// TwinCAT 3 PLC project UnloadRobot
// ProgramVersion: 3.1.4024.0
// libraries:
//   Tc2_EtherCAT, * (Beckhoff Automation GmbH)
//   Tc2_MC2, * (Beckhoff Automation GmbH)
//   Tc2_SerialCom, * (Beckhoff Automation GmbH)
//   Tc2_Standard, * (Beckhoff Automation GmbH)
//   Tc2_System, * (Beckhoff Automation GmbH)
//   Tc2_Utilities, * (Beckhoff Automation GmbH)
//   Tc3_Module, * (Beckhoff Automation GmbH)
// project tree:
//   DUTs/ Angles.TcDUT, Box.TcDUT, DUT.TcDUT, Points.TcDUT, SystemStatus.TcDUT
//   GVLs/ GVL_SerialComunication.TcGVL, Robot_Control_State.TcGVL, Robot_Motor.TcGVL, Robot_Parameter.TcGVL, Robot_Status_Info.TcGVL
//   / PlcTask.TcTTO
//   POUs/ AxisAllCtrl.TcPOU, AxisStatus.TcPOU, AxisStatusReadErrorCode.TcPOU, LedControl.TcPOU, LedLogic.TcPOU, TBoxCtrl.TcPOU, WheelCtrlButtonModeCheck.TcPOU, LeftArmFK.TcPOU, ArmFK_bak.TcPOU, LeftArmWristIK.TcPOU, MoveExtPos.TcPOU, RightArmManualCtrlMove.TcPOU, RightArmFK.TcPOU, LeftArmIK.TcPOU, ArmIK_bak.TcPOU, ArmMove.TcPOU, RightArmIK.TcPOU, LeftArmManualCtrlMove.TcPOU, AxisAbs.TcPOU, AxisCaliHomePos.TcPOU, AxisJog.TcPOU, AxisPowerOn.TcPOU, AxisReset.TcPOU, AxisStop.TcPOU, Gate_Back_Move.TcPOU, GateMove.TcPOU, Gate_Small_Move.TcPOU, MAIN.TcPOU, RightArmWristIK.TcPOU, WheelControl.TcPOU
//   POUs/Serial/ BmsSerial.TcPOU, BmsSerialBackground.TcPOU
// real-time tasks:
//   TASK PlcTask10ms: cycle T#10ms, priority 20, ADS port 350
// motion (NC):
//   TASK NC-Task 1 SAF: cycle T#2ms, priority 4, ADS port 501
//   TASK NC-Task 1 SVB: cycle T#10ms, priority 8, ADS port 511
//   AXIS Axis1_LeftArm_Left (id 3)
//     General: UnitName=°
//     Dynamic: Acceleration=100, Deceleration=150
//     Velo: RefSearch=5, RefSync=5, SlowManual=1, FastManual=5, Maximum=3000
//     OtherSettings: AllowMotionCmdToSlave=true, PulseDistancePos=1, PulseDistanceNeg=1
//     encoder EncType=19
//       EncPara: ScaleFactorNumerator=2.35294117647059, ScaleFactorDenominator=8388608, Offset=122.6484, MaxCount=#xffffffff, ReferenceSystem=1
//     drive DrvType=16
//       DrvPara: MaxCount=#xffffffff, DriveControlDWord=#x00020100
//         Analog: VeloReferenz=3300, TorqueSetpointScale=10, ScaleFactorActTorque=0.1
//         TimeComp: TaskDelayCycles=1
//     controller CtrType=1
//       CtrPara: PriorControlFactor=1
//         PosDiffControl: Enable=false
//         Observer: BandWidth=20
//   AXIS Axis2_LeftArm_Right (id 4)
//     General: UnitName=°
//     Dynamic: Acceleration=100
//     Velo: RefSearch=5, RefSync=5, SlowManual=1, FastManual=5, Maximum=3000
//     OtherSettings: AllowMotionCmdToSlave=true, PulseDistancePos=1, PulseDistanceNeg=1
//     encoder EncType=19
//       EncPara: ScaleFactorNumerator=2.35294117647059, ScaleFactorDenominator=8388608, Offset=68.5837, MaxCount=#xffffffff, ReferenceSystem=1
//     drive DrvType=16
//       DrvPara: MaxCount=#xffffffff, DriveControlDWord=#x00020100
//         Analog: VeloReferenz=3300, TorqueSetpointScale=10, ScaleFactorActTorque=0.1
//         TimeComp: TaskDelayCycles=1
//     controller CtrType=1
//       CtrPara: PriorControlFactor=1
//         PosDiffControl: Enable=false
//         Observer: BandWidth=20
//   AXIS Axis3_LeftArm_Wrist (id 5)
//     General: UnitName=°
//     Dynamic: Acceleration=30
//     Velo: RefSearch=5, RefSync=5, SlowManual=1, FastManual=5, Maximum=3000
//     OtherSettings: AllowMotionCmdToSlave=true, PulseDistancePos=1, PulseDistanceNeg=1
//     encoder EncType=19
//       EncPara: ScaleFactorNumerator=2.97520661157025, ScaleFactorDenominator=8388608, Offset=-19.23, MaxCount=#xffffffff, ReferenceSystem=1
//     drive DrvType=16
//       DrvPara: MaxCount=#xffffffff, DriveControlDWord=#x00020100
//         Analog: VeloReferenz=3300, TorqueSetpointScale=10, ScaleFactorActTorque=0.1
//         TimeComp: TaskDelayCycles=1
//     controller CtrType=1
//       CtrPara: PriorControlFactor=1
//         PosDiffControl: Enable=false
//         Observer: BandWidth=20
//   AXIS Axis4_LeftArm_Lift (id 9)
//     Dynamic: Acceleration=30
//     Velo: RefSearch=5, RefSync=5, SlowManual=1, FastManual=5, Maximum=3000
//     OtherSettings: AllowMotionCmdToSlave=true, PulseDistancePos=1, PulseDistanceNeg=1
//     encoder EncType=19
//       EncPara: ScaleFactorNumerator=6.03, ScaleFactorDenominator=8388608, Offset=-15.1688, MaxCount=#xffffffff, ReferenceSystem=1
//     drive DrvType=16
//       DrvPara: MaxCount=#xffffffff, DriveControlDWord=#x00020100
//         Analog: VeloReferenz=3300, TorqueSetpointScale=10, ScaleFactorActTorque=0.1
//         TimeComp: TaskDelayCycles=1
//     controller CtrType=1
//       CtrPara: PriorControlFactor=1
//         Observer: BandWidth=20
//   AXIS Axis5_RightArm_Left (id 6)
//     General: UnitName=°
//     Dynamic: Acceleration=100, Deceleration=100
//     Velo: RefSearch=5, RefSync=5, SlowManual=1, FastManual=5, Maximum=3000
//     OtherSettings: AllowMotionCmdToSlave=true, PulseDistancePos=1, PulseDistanceNeg=1
//     encoder EncType=19
//       EncPara: ScaleFactorNumerator=2.35294117647059, ScaleFactorDenominator=8388608, Offset=113, MaxCount=#xffffffff, ReferenceSystem=1
//     drive DrvType=16
//       DrvPara: MaxCount=#xffffffff, DriveControlDWord=#x00020100
//         Analog: VeloReferenz=3300, TorqueSetpointScale=10, ScaleFactorActTorque=0.1
//         TimeComp: TaskDelayCycles=1
//     controller CtrType=1
//       CtrPara: PriorControlFactor=1
//         PosDiffControl: Enable=false
//         Observer: BandWidth=20
//   AXIS Axis6_RightArm_Right (id 7)
//     General: UnitName=°
//     Dynamic: Acceleration=100, Deceleration=100
//     Velo: RefSearch=5, RefSync=5, SlowManual=1, FastManual=5, Maximum=3000
//     OtherSettings: AllowMotionCmdToSlave=true, PulseDistancePos=1, PulseDistanceNeg=1
//     encoder EncType=19
//       EncPara: ScaleFactorNumerator=2.35294117647059, ScaleFactorDenominator=8388608, Offset=58, MaxCount=#xffffffff, ReferenceSystem=1
//     drive DrvType=16
//       DrvPara: MaxCount=#xffffffff, DriveControlDWord=#x00020100
//         Analog: VeloReferenz=3300, TorqueSetpointScale=10, ScaleFactorActTorque=0.1
//         TimeComp: TaskDelayCycles=1
//     controller CtrType=1
//       CtrPara: PriorControlFactor=1
//         PosDiffControl: Enable=false
//         Observer: BandWidth=20
//   AXIS Axis7_RightArm_Wrist (id 8)
//     General: UnitName=°
//     Dynamic: Acceleration=30
//     Velo: RefSearch=5, RefSync=5, SlowManual=1, FastManual=5, Maximum=3000
//     OtherSettings: AllowMotionCmdToSlave=true, PulseDistancePos=1, PulseDistanceNeg=1
//     encoder EncType=19
//       EncPara: ScaleFactorNumerator=2.97520661157025, ScaleFactorDenominator=8388608, Offset=24.6504, MaxCount=#xffffffff, ReferenceSystem=1
//     drive DrvType=16
//       DrvPara: MaxCount=#xffffffff, DriveControlDWord=#x00020100
//         Analog: VeloReferenz=3300, TorqueSetpointScale=10, ScaleFactorActTorque=0.1
//         TimeComp: TaskDelayCycles=1
//     controller CtrType=1
//       CtrPara: PriorControlFactor=1
//         Observer: BandWidth=20
//   AXIS Axis8_RightArm_Lift (id 10)
//     Dynamic: Acceleration=30
//     Velo: RefSearch=5, RefSync=5, SlowManual=1, FastManual=5, Maximum=3000
//     OtherSettings: AllowMotionCmdToSlave=true, PulseDistancePos=1, PulseDistanceNeg=1
//     encoder EncType=19
//       EncPara: ScaleFactorNumerator=6.03, ScaleFactorDenominator=8388608, Offset=5.5077, MaxCount=#xffffffff, ReferenceSystem=1
//     drive DrvType=16
//       DrvPara: MaxCount=#xffffffff, DriveControlDWord=#x00020100
//         Analog: VeloReferenz=3300, TorqueSetpointScale=10, ScaleFactorActTorque=0.1
//         TimeComp: TaskDelayCycles=1
//     controller CtrType=1
//       CtrPara: PriorControlFactor=1
//         Observer: BandWidth=20
//   AXIS Axis9_BigGate_Left (id 11)
//     Dynamic: Acceleration=101, Deceleration=109.503, Jerk=510.05
//     Velo: RefSearch=5, RefSync=5, SlowManual=1, FastManual=5
//     OtherSettings: AllowMotionCmdToSlave=true, PulseDistancePos=1, PulseDistanceNeg=1
//     encoder EncType=19
//       EncPara: ScaleFactorNumerator=6.03, ScaleFactorDenominator=8388608, Offset=361.3851, MaxCount=#xffffffff, ReferenceSystem=1
//         SoftEndMinControl: Enable=true, Range=-5
//         SoftEndMaxControl: Enable=true, Range=860
//     drive DrvType=16
//       DrvPara: MaxCount=#xffffffff, DriveControlDWord=#x00020100
//         Analog: TorqueSetpointScale=10, ScaleFactorActTorque=0.1
//         TimeComp: TaskDelayCycles=1
//     controller CtrType=1
//       CtrPara: PriorControlFactor=1
//         Observer: BandWidth=20
//   AXIS Axis10_BigGate_Right (id 12)
//     Dynamic: Acceleration=101, Deceleration=108.497, Jerk=510.05
//     Velo: RefSearch=5, RefSync=5, SlowManual=1, FastManual=5
//     OtherSettings: AllowMotionCmdToSlave=true, PulseDistancePos=1, PulseDistanceNeg=1
//     encoder EncType=19
//       EncPara: ScaleFactorNumerator=6.03, ScaleFactorDenominator=8388608, Offset=-371.0742, MaxCount=#xffffffff, ReferenceSystem=1
//         SoftEndMinControl: Enable=true, Range=-860
//         SoftEndMaxControl: Enable=true, Range=5
//     drive DrvType=16
//       DrvPara: MaxCount=#xffffffff, DriveControlDWord=#x00020100
//         Analog: TorqueSetpointScale=10, ScaleFactorActTorque=0.1
//         TimeComp: TaskDelayCycles=1
//     controller CtrType=1
//       CtrPara: PriorControlFactor=1
//         Observer: BandWidth=20
//   AXIS Axis11_SmallGate_Left (id 13)
//     Dynamic: Acceleration=100
//     Velo: RefSearch=5, RefSync=5, SlowManual=1, FastManual=5
//     OtherSettings: AllowMotionCmdToSlave=true, PulseDistancePos=1, PulseDistanceNeg=1
//     encoder EncType=19
//       EncPara: ScaleFactorNumerator=6.03, ScaleFactorDenominator=8388608, Offset=23.9905, MaxCount=#xffffffff, ReferenceSystem=1
//         SoftEndMinControl: Enable=true, Range=-980
//         SoftEndMaxControl: Enable=true, Range=5
//     drive DrvType=16
//       DrvPara: MaxCount=#xffffffff, DriveControlDWord=#x00020100
//         Analog: TorqueSetpointScale=10, ScaleFactorActTorque=0.1
//         TimeComp: TaskDelayCycles=1
//     controller CtrType=1
//       CtrPara: PriorControlFactor=1
//         Observer: BandWidth=20
//   AXIS Axis12_SmallGate_Right (id 14)
//     Dynamic: Acceleration=100
//     Velo: RefSearch=5, RefSync=5, SlowManual=1, FastManual=5
//     OtherSettings: AllowMotionCmdToSlave=true, PulseDistancePos=1, PulseDistanceNeg=1
//     encoder EncType=19
//       EncPara: ScaleFactorNumerator=6.03, ScaleFactorDenominator=8388608, Offset=-28.5893, MaxCount=#xffffffff, ReferenceSystem=1
//         SoftEndMinControl: Enable=true, Range=-5
//         SoftEndMaxControl: Enable=true, Range=980
//     drive DrvType=16
//       DrvPara: MaxCount=#xffffffff, DriveControlDWord=#x00020100
//         Analog: TorqueSetpointScale=10, ScaleFactorActTorque=0.1
//         TimeComp: TaskDelayCycles=1
//     controller CtrType=1
//       CtrPara: PriorControlFactor=1
//         Observer: BandWidth=20
//   AXIS Axis13_BackGate_Left (id 15)
//     Dynamic: Acceleration=100
//     Velo: RefSearch=5, RefSync=5, SlowManual=1, FastManual=5, Maximum=3000
//     OtherSettings: AllowMotionCmdToSlave=true, PulseDistancePos=1, PulseDistanceNeg=1
//     encoder EncType=19
//       EncPara: ScaleFactorNumerator=5, ScaleFactorDenominator=8388608, Offset=-120.0448, MaxCount=#xffffffff, ReferenceSystem=1
//         SoftEndMinControl: Enable=true, Range=-300
//     drive DrvType=16
//       DrvPara: MaxCount=#xffffffff, DriveControlDWord=#x00020100
//         Analog: VeloReferenz=3300, TorqueSetpointScale=10, ScaleFactorActTorque=0.1
//         TimeComp: TaskDelayCycles=1
//     controller CtrType=1
//       CtrPara: PriorControlFactor=1
//         Observer: BandWidth=20
//   AXIS Axis14_BackGate_Right (id 16)
//     Dynamic: Acceleration=100
//     Velo: RefSearch=5, RefSync=5, SlowManual=1, FastManual=5, Maximum=3000
//     OtherSettings: AllowMotionCmdToSlave=true, PulseDistancePos=1, PulseDistanceNeg=1
//     encoder EncType=19
//       EncPara: ScaleFactorNumerator=5, ScaleFactorDenominator=8388608, Offset=-44.1864, MaxCount=#xffffffff, ReferenceSystem=1
//         SoftEndMinControl: Enable=true, Range=-300
//     drive DrvType=16
//       DrvPara: MaxCount=#xffffffff, DriveControlDWord=#x00020100
//         Analog: VeloReferenz=3300, TorqueSetpointScale=10, ScaleFactorActTorque=0.1
//         TimeComp: TaskDelayCycles=1
//     controller CtrType=1
//       CtrPara: PriorControlFactor=1
//         Observer: BandWidth=20
//   AXIS Axis15_RightWheel_Steer (id 18)
//     General: UnitName=°
//     Velo: RefSearch=2, RefSync=2, SlowManual=5, FastManual=10, Maximum=3000
//     OtherSettings: AllowMotionCmdToSlave=true
//     encoder EncType=19
//       EncPara: ScaleFactorNumerator=1.14285714285714, ScaleFactorDenominator=65535, Offset=-120, MaxCount=#xffffffff, ReferenceSystem=1
//     drive DrvType=16
//       DrvPara: MaxCount=#xffffffff, DriveControlDWord=#x00020000
//         Analog: VeloReferenz=3300, TorqueSetpointScale=10, ScaleFactorActTorque=0.1
//         TimeComp: TaskDelayCycles=1
//     controller CtrType=1
//       CtrPara: PriorControlFactor=1
//         PosDiffControl: Enable=false
//         Observer: BandWidth=20
//   AXIS Axis16_RightWheel_Walk (id 19)
//     Dynamic: AccelerationMaximum=1334, DecelerationMaximum=1334, Acceleration=999.99950000025, Deceleration=999.99950000025, Jerk=1000.00100000175
//     Velo: RefSearch=5, RefSync=5, SlowManual=30, FastManual=60, Maximum=3000
//     OtherSettings: AllowMotionCmdToSlave=true
//     encoder EncType=19
//       EncPara: ScaleFactorNumerator=17.27, ScaleFactorDenominator=65535, MaxCount=#xffffffff
//     drive DrvType=16
//       DrvPara: MaxCount=#xffffffff, DriveControlDWord=#x00020000
//         Analog: VeloReferenz=3300, TorqueSetpointScale=10, ScaleFactorActTorque=0.1
//         TimeComp: TaskDelayCycles=1
//     controller CtrType=1
//       CtrPara: PriorControlFactor=1
//         PosDiffControl: Enable=false
//         Observer: BandWidth=20
//   AXIS Axis17_LeftWheel_Steer (id 20)
//     General: UnitName=°
//     Velo: RefSearch=2, RefSync=2, SlowManual=5, FastManual=10
//     OtherSettings: AllowMotionCmdToSlave=true
//     encoder EncType=19
//       EncPara: ScaleFactorNumerator=1.14285714285714, ScaleFactorDenominator=65535, Offset=-120, MaxCount=#xffffffff, ReferenceSystem=1
//     drive DrvType=16
//       DrvPara: MaxCount=#xffffffff, DriveControlDWord=#x00020000
//         Analog: TorqueSetpointScale=10, ScaleFactorActTorque=0.1
//         TimeComp: TaskDelayCycles=1
//     controller CtrType=1
//       CtrPara: PriorControlFactor=1
//         PosDiffControl: Enable=false
//         Observer: BandWidth=20
//   AXIS Axis18_LeftWheel_Walk (id 21)
//     Dynamic: AccelerationMaximum=1334, DecelerationMaximum=1334, Acceleration=999.998, Deceleration=999.998, Jerk=1000
//     Velo: RefSearch=5, RefSync=5, SlowManual=30, FastManual=60, Maximum=3000
//     OtherSettings: AllowMotionCmdToSlave=true
//     encoder EncType=19
//       EncPara: ScaleFactorNumerator=17.27, ScaleFactorDenominator=65535, MaxCount=#xffffffff
//     drive DrvType=16
//       DrvPara: MaxCount=#xffffffff, DriveControlDWord=#x00020000
//         Analog: VeloReferenz=3300, TorqueSetpointScale=10, ScaleFactorActTorque=0.1
//         TimeComp: TaskDelayCycles=1
//     controller CtrType=1
//       CtrPara: PriorControlFactor=1
//         PosDiffControl: Enable=false
//         Observer: BandWidth=20
//   AXIS Axis01_TestArm_Right (id 1)
//     General: UnitName=°
//     Dynamic: Acceleration=100
//     Velo: Maximum=3000
//     OtherSettings: AllowMotionCmdToSlave=true
//     encoder EncType=1
//       EncPara: ScaleFactorNumerator=360, ScaleFactorDenominator=8388608, Offset=-210.5505, ReferenceSystem=1
//         SoftEndMinControl: Enable=true, Range=-40
//         SoftEndMaxControl: Enable=true, Range=130
//     drive DrvType=5
//       Analog: VeloReferenz=3300, TorqueSetpointScale=10, ScaleFactorActTorque=0.1
//       TimeComp: TaskDelayCycles=1
//     controller CtrType=1
//       CtrPara: PriorControlFactor=1
//         Observer: BandWidth=20
//   AXIS Axis02_TestArm_Left (id 2)
//     General: UnitName=°
//     Dynamic: Acceleration=100.851, Jerk=339.029
//     Velo: Maximum=3000
//     OtherSettings: AllowMotionCmdToSlave=true
//     encoder EncType=19
//       EncPara: ScaleFactorNumerator=360, ScaleFactorDenominator=8388608, Offset=225.616, MaxCount=#xffffffff, ReferenceSystem=1
//         SoftEndMinControl: Enable=true, Range=40
//         SoftEndMaxControl: Enable=true, Range=220
//     drive DrvType=16
//       DrvPara: MaxCount=#xffffffff, DriveControlDWord=#x00000100
//         Analog: VeloReferenz=3300, TorqueSetpointScale=10, ScaleFactorActTorque=0.1
//         TimeComp: TaskDelayCycles=1
//     controller CtrType=1
//       CtrPara: PriorControlFactor=1
//         Observer: BandWidth=20
//   AXIS Axis03_TestArm_Wrist (id 17)
//     General: UnitName=°
//     Dynamic: Acceleration=100.851, Jerk=339.029
//     Velo: Maximum=3000
//     OtherSettings: AllowMotionCmdToSlave=true
//     encoder EncType=19
//       EncPara: ScaleFactorNumerator=360, ScaleFactorDenominator=8388608, Offset=225.616, MaxCount=#xffffffff, ReferenceSystem=1
//         SoftEndMinControl: Enable=true, Range=40
//         SoftEndMaxControl: Enable=true, Range=220
//     drive DrvType=16
//       DrvPara: MaxCount=#xffffffff, DriveControlDWord=#x00000100
//         Analog: VeloReferenz=3300, TorqueSetpointScale=10, ScaleFactorActTorque=0.1
//         TimeComp: TaskDelayCycles=1
//     controller CtrType=1
//       CtrPara: PriorControlFactor=1
//         Observer: BandWidth=20
// I/O:
//   DEVICE Device 3 (EtherCAT), AmsNetId 192.168.1.20.2.1
//     Term 8 (EK1200) [EK1200-5000 EtherCAT Power supply (2A E-Bus)]
//       Term 17 (EL1809) [EL1809 16Ch. Dig. Input 24V, 3ms]
//       Term 18 (EL1809) [EL1809 16Ch. Dig. Input 24V, 3ms]
//       Term 19 (EL1809) [EL1809 16Ch. Dig. Input 24V, 3ms]
//       Term 20 (EL2809) [EL2809 16Ch. Dig. Output 24V, 0.5A]
//       Term 21 (EL2809) [EL2809 16Ch. Dig. Output 24V, 0.5A]
//       Term 24 (EK1110) [EK1110 EtherCAT extension]
//     Drive RightWheel Steer (XMC_ESC) [XMC_ESC]
//     Drive RightWheel Walk (XMC_ESC) [XMC_ESC]
//     Drive LeftWheel Steer (XMC_ESC) [XMC_ESC]
//     Drive LeftWheel Walk (XMC_ESC) [XMC_ESC]
//   DEVICE Device 4 (EtherCAT), AmsNetId 192.168.1.20.5.1
//     Drive BackGate Right(MCDLN35BE) [MCDLN35BE]
//     Drive RightArm Wrist (MBDLN25BE) [MBDLN25BE]
//     Drive RightArm Left (MDDLN55BE) [MDDLN55BE]
//     Drive RightArm Lift (MDDLN55BE) [MDDLN55BE]
//     Drive RightArm Right (MDDLN55BE) [MDDLN55BE]
//     Drive SmallGate Right (MDDLN45BE) [MDDLN45BE]
//     Drive BigGate Right (MDDLN55BE) [MDDLN55BE]
//     Drive BackGate Left (MCDLN35BE) [MCDLN35BE]
//     Drive BigGate Left (MDDLN55BE) [MDDLN55BE]
//     Drive SmallGate Left (MDDLN45BE) [MDDLN45BE]
//     Drive LeftArm Lift (MDDLN55BE) [MDDLN55BE]
//     Drive LeftArm Right (MDDLN55BE) [MDDLN55BE]
//     Drive LeftArm Wrist (MBDLN25BE) [MBDLN25BE]
//     Drive LeftArm Left (MDDLN55BE) [MDDLN55BE]
//   DEVICE Device 5 (COM Port)
//   DEVICE Device 6 (NOV-DP-RAM)
//   DEVICE Device 3 (EtherCAT Automation Protocol), AmsNetId 192.168.1.20.4.1
//   DEVICE Device 7 (USB)
//     Box 1 (CX2100 Power Supply)
// variable links:
//   NC-Task 1 SAF/Axes/Axis10_BigGate_Right <-> Device 4 (EtherCAT)/Drive BigGate Right (MDDLN55BE)
//     Drive/Inputs/In/nDataIn1 <-> Transmit PDO mapping 1/Following error actual value
//     Drive/Inputs/In/nDataIn3[0] <-> Transmit PDO mapping 1/Torque actual value
//     Drive/Inputs/In/nDcOutputTime <-> InfoData/DcOutputShift
//     Drive/Inputs/In/nState1 <-> Transmit PDO mapping 1/Statusword
//     Drive/Inputs/In/nState2 <-> Transmit PDO mapping 1/Statusword @bit 8
//     Drive/Inputs/In/nState4 @bit 1 <-> WcState/InputToggle
//     Drive/Inputs/In/nState4 <-> WcState/WcState
//     Drive/Inputs/In/nState5 <-> Transmit PDO mapping 1/Modes of operation display
//     Drive/Outputs/Out/nCtrl1 <-> Receive PDO mapping 1/Controlword
//     Drive/Outputs/Out/nCtrl2 <-> Receive PDO mapping 1/Controlword @bit 8
//     Drive/Outputs/Out/nCtrl5 <-> Receive PDO mapping 1/Modes of operation
//     Drive/Outputs/Out/nDataOut1 <-> Receive PDO mapping 1/Target position
//     Enc/Inputs/In/nDataIn1 <-> Transmit PDO mapping 1/Position actual value
//     Enc/Inputs/In/nDataIn3 <-> Transmit PDO mapping 1/Touch probe pos1 pos value
//     Enc/Inputs/In/nDcInputTime <-> InfoData/DcInputShift
//     Enc/Inputs/In/nState4 @bit 1 <-> WcState/InputToggle
//     Enc/Inputs/In/nState4 <-> WcState/WcState
//     Enc/Inputs/In/nState5 <-> Transmit PDO mapping 1/Touch probe status
//     Enc/Inputs/In/nState6 <-> Transmit PDO mapping 1/Touch probe status @bit 8
//     Enc/Outputs/Out/nCtrl5 <-> Receive PDO mapping 1/Touch probe function
//     Enc/Outputs/Out/nCtrl6 <-> Receive PDO mapping 1/Touch probe function @bit 8
//   NC-Task 1 SAF/Axes/Axis11_SmallGate_Left <-> Device 4 (EtherCAT)/Drive SmallGate Left (MDDLN45BE)
//     Drive/Inputs/In/nDataIn1 <-> Transmit PDO mapping 1/Following error actual value
//     Drive/Inputs/In/nDataIn3[0] <-> Transmit PDO mapping 1/Torque actual value
//     Drive/Inputs/In/nDcOutputTime <-> InfoData/DcOutputShift
//     Drive/Inputs/In/nState1 <-> Transmit PDO mapping 1/Statusword
//     Drive/Inputs/In/nState2 <-> Transmit PDO mapping 1/Statusword @bit 8
//     Drive/Inputs/In/nState4 @bit 1 <-> WcState/InputToggle
//     Drive/Inputs/In/nState4 <-> WcState/WcState
//     Drive/Inputs/In/nState5 <-> Transmit PDO mapping 1/Modes of operation display
//     Drive/Outputs/Out/nCtrl1 <-> Receive PDO mapping 1/Controlword
//     Drive/Outputs/Out/nCtrl2 <-> Receive PDO mapping 1/Controlword @bit 8
//     Drive/Outputs/Out/nCtrl5 <-> Receive PDO mapping 1/Modes of operation
//     Drive/Outputs/Out/nDataOut1 <-> Receive PDO mapping 1/Target position
//     Enc/Inputs/In/nDataIn1 <-> Transmit PDO mapping 1/Position actual value
//     Enc/Inputs/In/nDataIn3 <-> Transmit PDO mapping 1/Touch probe pos1 pos value
//     Enc/Inputs/In/nDcInputTime <-> InfoData/DcInputShift
//     Enc/Inputs/In/nState4 @bit 1 <-> WcState/InputToggle
//     Enc/Inputs/In/nState4 <-> WcState/WcState
//     Enc/Inputs/In/nState5 <-> Transmit PDO mapping 1/Touch probe status
//     Enc/Inputs/In/nState6 <-> Transmit PDO mapping 1/Touch probe status @bit 8
//     Enc/Outputs/Out/nCtrl5 <-> Receive PDO mapping 1/Touch probe function
//     Enc/Outputs/Out/nCtrl6 <-> Receive PDO mapping 1/Touch probe function @bit 8
//   NC-Task 1 SAF/Axes/Axis12_SmallGate_Right <-> Device 4 (EtherCAT)/Drive SmallGate Right (MDDLN45BE)
//     Drive/Inputs/In/nDataIn1 <-> Transmit PDO mapping 1/Following error actual value
//     Drive/Inputs/In/nDataIn3[0] <-> Transmit PDO mapping 1/Torque actual value
//     Drive/Inputs/In/nDcOutputTime <-> InfoData/DcOutputShift
//     Drive/Inputs/In/nState1 <-> Transmit PDO mapping 1/Statusword
//     Drive/Inputs/In/nState2 <-> Transmit PDO mapping 1/Statusword @bit 8
//     Drive/Inputs/In/nState4 @bit 1 <-> WcState/InputToggle
//     Drive/Inputs/In/nState4 <-> WcState/WcState
//     Drive/Inputs/In/nState5 <-> Transmit PDO mapping 1/Modes of operation display
//     Drive/Outputs/Out/nCtrl1 <-> Receive PDO mapping 1/Controlword
//     Drive/Outputs/Out/nCtrl2 <-> Receive PDO mapping 1/Controlword @bit 8
//     Drive/Outputs/Out/nCtrl5 <-> Receive PDO mapping 1/Modes of operation
//     Drive/Outputs/Out/nDataOut1 <-> Receive PDO mapping 1/Target position
//     Enc/Inputs/In/nDataIn1 <-> Transmit PDO mapping 1/Position actual value
//     Enc/Inputs/In/nDataIn3 <-> Transmit PDO mapping 1/Touch probe pos1 pos value
//     Enc/Inputs/In/nDcInputTime <-> InfoData/DcInputShift
//     Enc/Inputs/In/nState4 @bit 1 <-> WcState/InputToggle
//     Enc/Inputs/In/nState4 <-> WcState/WcState
//     Enc/Inputs/In/nState5 <-> Transmit PDO mapping 1/Touch probe status
//     Enc/Inputs/In/nState6 <-> Transmit PDO mapping 1/Touch probe status @bit 8
//     Enc/Outputs/Out/nCtrl5 <-> Receive PDO mapping 1/Touch probe function
//     Enc/Outputs/Out/nCtrl6 <-> Receive PDO mapping 1/Touch probe function @bit 8
//   NC-Task 1 SAF/Axes/Axis13_BackGate_Left <-> Device 4 (EtherCAT)/Drive BackGate Left (MCDLN35BE)
//     Drive/Inputs/In/nDataIn1 <-> Transmit PDO mapping 1/Following error actual value
//     Drive/Inputs/In/nDataIn3[0] <-> Transmit PDO mapping 1/Torque actual value
//     Drive/Inputs/In/nDcOutputTime <-> InfoData/DcOutputShift
//     Drive/Inputs/In/nState1 <-> Transmit PDO mapping 1/Statusword
//     Drive/Inputs/In/nState2 <-> Transmit PDO mapping 1/Statusword @bit 8
//     Drive/Inputs/In/nState4 @bit 1 <-> WcState/InputToggle
//     Drive/Inputs/In/nState4 <-> WcState/WcState
//     Drive/Inputs/In/nState5 <-> Transmit PDO mapping 1/Modes of operation display
//     Drive/Outputs/Out/nCtrl1 <-> Receive PDO mapping 1/Controlword
//     Drive/Outputs/Out/nCtrl2 <-> Receive PDO mapping 1/Controlword @bit 8
//     Drive/Outputs/Out/nCtrl5 <-> Receive PDO mapping 1/Modes of operation
//     Drive/Outputs/Out/nDataOut1 <-> Receive PDO mapping 1/Target position
//     Enc/Inputs/In/nDataIn1 <-> Transmit PDO mapping 1/Position actual value
//     Enc/Inputs/In/nDataIn3 <-> Transmit PDO mapping 1/Touch probe pos1 pos value
//     Enc/Inputs/In/nDcInputTime <-> InfoData/DcInputShift
//     Enc/Inputs/In/nState4 @bit 1 <-> WcState/InputToggle
//     Enc/Inputs/In/nState4 <-> WcState/WcState
//     Enc/Inputs/In/nState5 <-> Transmit PDO mapping 1/Touch probe status
//     Enc/Inputs/In/nState6 <-> Transmit PDO mapping 1/Touch probe status @bit 8
//     Enc/Outputs/Out/nCtrl5 <-> Receive PDO mapping 1/Touch probe function
//     Enc/Outputs/Out/nCtrl6 <-> Receive PDO mapping 1/Touch probe function @bit 8
//   NC-Task 1 SAF/Axes/Axis14_BackGate_Right <-> Device 4 (EtherCAT)/Drive BackGate Right(MCDLN35BE)
//     Drive/Inputs/In/nDataIn1 <-> Transmit PDO mapping 1/Following error actual value
//     Drive/Inputs/In/nDataIn3[0] <-> Transmit PDO mapping 1/Torque actual value
//     Drive/Inputs/In/nDcOutputTime <-> InfoData/DcOutputShift
//     Drive/Inputs/In/nState1 <-> Transmit PDO mapping 1/Statusword
//     Drive/Inputs/In/nState2 <-> Transmit PDO mapping 1/Statusword @bit 8
//     Drive/Inputs/In/nState4 @bit 1 <-> WcState/InputToggle
//     Drive/Inputs/In/nState4 <-> WcState/WcState
//     Drive/Inputs/In/nState5 <-> Transmit PDO mapping 1/Modes of operation display
//     Drive/Outputs/Out/nCtrl1 <-> Receive PDO mapping 1/Controlword
//     Drive/Outputs/Out/nCtrl2 <-> Receive PDO mapping 1/Controlword @bit 8
//     Drive/Outputs/Out/nCtrl5 <-> Receive PDO mapping 1/Modes of operation
//     Drive/Outputs/Out/nDataOut1 <-> Receive PDO mapping 1/Target position
//     Enc/Inputs/In/nDataIn1 <-> Transmit PDO mapping 1/Position actual value
//     Enc/Inputs/In/nDataIn3 <-> Transmit PDO mapping 1/Touch probe pos1 pos value
//     Enc/Inputs/In/nDcInputTime <-> InfoData/DcInputShift
//     Enc/Inputs/In/nState4 @bit 1 <-> WcState/InputToggle
//     Enc/Inputs/In/nState4 <-> WcState/WcState
//     Enc/Inputs/In/nState5 <-> Transmit PDO mapping 1/Touch probe status
//     Enc/Inputs/In/nState6 <-> Transmit PDO mapping 1/Touch probe status @bit 8
//     Enc/Outputs/Out/nCtrl5 <-> Receive PDO mapping 1/Touch probe function
//     Enc/Outputs/Out/nCtrl6 <-> Receive PDO mapping 1/Touch probe function @bit 8
//   NC-Task 1 SAF/Axes/Axis15_RightWheel_Steer <-> Device 3 (EtherCAT)/Drive RightWheel Steer (XMC_ESC)
//     Drive/Inputs/In/nState1 <-> TxPDO/Statusword
//     Drive/Inputs/In/nState2 <-> TxPDO/Statusword
//     Drive/Outputs/Out/nCtrl1 <-> RxPDO/Controlword
//     Drive/Outputs/Out/nDataOut1 <-> RxPDO/Target_position
//     Enc/Inputs/In/nDataIn1 <-> TxPDO/Position actual angle vaule
//   NC-Task 1 SAF/Axes/Axis16_RightWheel_Walk <-> Device 3 (EtherCAT)/Drive RightWheel Walk (XMC_ESC)
//     Drive/Inputs/In/nState1 <-> TxPDO/Statusword
//     Drive/Inputs/In/nState2 <-> TxPDO/Statusword
//     Drive/Outputs/Out/nCtrl1 <-> RxPDO/Controlword
//     Drive/Outputs/Out/nDataOut1 <-> RxPDO/Target_position
//     Enc/Inputs/In/nDataIn1 <-> TxPDO/Position actual angle vaule
//   NC-Task 1 SAF/Axes/Axis17_LeftWheel_Steer <-> Device 3 (EtherCAT)/Drive LeftWheel Steer (XMC_ESC)
//     Drive/Inputs/In/nState1 <-> TxPDO/Statusword
//     Drive/Inputs/In/nState2 <-> TxPDO/Statusword
//     Drive/Outputs/Out/nCtrl1 <-> RxPDO/Controlword
//     Drive/Outputs/Out/nDataOut1 <-> RxPDO/Target_position
//     Enc/Inputs/In/nDataIn1 <-> TxPDO/Position actual angle vaule
//   NC-Task 1 SAF/Axes/Axis18_LeftWheel_Walk <-> Device 3 (EtherCAT)/Drive LeftWheel Walk (XMC_ESC)
//     Drive/Inputs/In/nState1 <-> TxPDO/Statusword
//     Drive/Inputs/In/nState2 <-> TxPDO/Statusword
//     Drive/Outputs/Out/nCtrl1 <-> RxPDO/Controlword
//     Drive/Outputs/Out/nDataOut1 <-> RxPDO/Target_position
//     Enc/Inputs/In/nDataIn1 <-> TxPDO/Position actual angle vaule
//   NC-Task 1 SAF/Axes/Axis1_LeftArm_Left <-> Device 4 (EtherCAT)/Drive LeftArm Left (MDDLN55BE)
//     Drive/Inputs/In/nDataIn1 <-> Transmit PDO mapping 1/Following error actual value
//     Drive/Inputs/In/nDataIn3[0] <-> Transmit PDO mapping 1/Torque actual value
//     Drive/Inputs/In/nDcOutputTime <-> InfoData/DcOutputShift
//     Drive/Inputs/In/nState1 <-> Transmit PDO mapping 1/Statusword
//     Drive/Inputs/In/nState2 <-> Transmit PDO mapping 1/Statusword @bit 8
//     Drive/Inputs/In/nState4 @bit 1 <-> WcState/InputToggle
//     Drive/Inputs/In/nState4 <-> WcState/WcState
//     Drive/Inputs/In/nState5 <-> Transmit PDO mapping 1/Modes of operation display
//     Drive/Outputs/Out/nCtrl1 <-> Receive PDO mapping 1/Controlword
//     Drive/Outputs/Out/nCtrl2 <-> Receive PDO mapping 1/Controlword @bit 8
//     Drive/Outputs/Out/nCtrl5 <-> Receive PDO mapping 1/Modes of operation
//     Drive/Outputs/Out/nDataOut1 <-> Receive PDO mapping 1/Target position
//     Enc/Inputs/In/nDataIn1 <-> Transmit PDO mapping 1/Position actual value
//     Enc/Inputs/In/nDataIn3 <-> Transmit PDO mapping 1/Touch probe pos1 pos value
//     Enc/Inputs/In/nDcInputTime <-> InfoData/DcInputShift
//     Enc/Inputs/In/nState4 @bit 1 <-> WcState/InputToggle
//     Enc/Inputs/In/nState4 <-> WcState/WcState
//     Enc/Inputs/In/nState5 <-> Transmit PDO mapping 1/Touch probe status
//     Enc/Inputs/In/nState6 <-> Transmit PDO mapping 1/Touch probe status @bit 8
//     Enc/Outputs/Out/nCtrl5 <-> Receive PDO mapping 1/Touch probe function
//     Enc/Outputs/Out/nCtrl6 <-> Receive PDO mapping 1/Touch probe function @bit 8
//   NC-Task 1 SAF/Axes/Axis2_LeftArm_Right <-> Device 4 (EtherCAT)/Drive LeftArm Right (MDDLN55BE)
//     Drive/Inputs/In/nDataIn1 <-> Transmit PDO mapping 1/Following error actual value
//     Drive/Inputs/In/nDataIn3[0] <-> Transmit PDO mapping 1/Torque actual value
//     Drive/Inputs/In/nDcOutputTime <-> InfoData/DcOutputShift
//     Drive/Inputs/In/nState1 <-> Transmit PDO mapping 1/Statusword
//     Drive/Inputs/In/nState2 <-> Transmit PDO mapping 1/Statusword @bit 8
//     Drive/Inputs/In/nState4 @bit 1 <-> WcState/InputToggle
//     Drive/Inputs/In/nState4 <-> WcState/WcState
//     Drive/Inputs/In/nState5 <-> Transmit PDO mapping 1/Modes of operation display
//     Drive/Outputs/Out/nCtrl1 <-> Receive PDO mapping 1/Controlword
//     Drive/Outputs/Out/nCtrl2 <-> Receive PDO mapping 1/Controlword @bit 8
//     Drive/Outputs/Out/nCtrl5 <-> Receive PDO mapping 1/Modes of operation
//     Drive/Outputs/Out/nDataOut1 <-> Receive PDO mapping 1/Target position
//     Enc/Inputs/In/nDataIn1 <-> Transmit PDO mapping 1/Position actual value
//     Enc/Inputs/In/nDataIn3 <-> Transmit PDO mapping 1/Touch probe pos1 pos value
//     Enc/Inputs/In/nDcInputTime <-> InfoData/DcInputShift
//     Enc/Inputs/In/nState4 @bit 1 <-> WcState/InputToggle
//     Enc/Inputs/In/nState4 <-> WcState/WcState
//     Enc/Inputs/In/nState5 <-> Transmit PDO mapping 1/Touch probe status
//     Enc/Inputs/In/nState6 <-> Transmit PDO mapping 1/Touch probe status @bit 8
//     Enc/Outputs/Out/nCtrl5 <-> Receive PDO mapping 1/Touch probe function
//     Enc/Outputs/Out/nCtrl6 <-> Receive PDO mapping 1/Touch probe function @bit 8
//   NC-Task 1 SAF/Axes/Axis3_LeftArm_Wrist <-> Device 4 (EtherCAT)/Drive LeftArm Wrist (MBDLN25BE)
//     Drive/Inputs/In/nDataIn1 <-> Transmit PDO mapping 1/Following error actual value
//     Drive/Inputs/In/nDataIn3[0] <-> Transmit PDO mapping 1/Torque actual value
//     Drive/Inputs/In/nDcOutputTime <-> InfoData/DcOutputShift
//     Drive/Inputs/In/nState1 <-> Transmit PDO mapping 1/Statusword
//     Drive/Inputs/In/nState2 <-> Transmit PDO mapping 1/Statusword @bit 8
//     Drive/Inputs/In/nState4 @bit 1 <-> WcState/InputToggle
//     Drive/Inputs/In/nState4 <-> WcState/WcState
//     Drive/Inputs/In/nState5 <-> Transmit PDO mapping 1/Modes of operation display
//     Drive/Outputs/Out/nCtrl1 <-> Receive PDO mapping 1/Controlword
//     Drive/Outputs/Out/nCtrl2 <-> Receive PDO mapping 1/Controlword @bit 8
//     Drive/Outputs/Out/nCtrl5 <-> Receive PDO mapping 1/Modes of operation
//     Drive/Outputs/Out/nDataOut1 <-> Receive PDO mapping 1/Target position
//     Enc/Inputs/In/nDataIn1 <-> Transmit PDO mapping 1/Position actual value
//     Enc/Inputs/In/nDataIn3 <-> Transmit PDO mapping 1/Touch probe pos1 pos value
//     Enc/Inputs/In/nDcInputTime <-> InfoData/DcInputShift
//     Enc/Inputs/In/nState4 @bit 1 <-> WcState/InputToggle
//     Enc/Inputs/In/nState4 <-> WcState/WcState
//     Enc/Inputs/In/nState5 <-> Transmit PDO mapping 1/Touch probe status
//     Enc/Inputs/In/nState6 <-> Transmit PDO mapping 1/Touch probe status @bit 8
//     Enc/Outputs/Out/nCtrl5 <-> Receive PDO mapping 1/Touch probe function
//     Enc/Outputs/Out/nCtrl6 <-> Receive PDO mapping 1/Touch probe function @bit 8
//   NC-Task 1 SAF/Axes/Axis4_LeftArm_Lift <-> Device 4 (EtherCAT)/Drive LeftArm Lift (MDDLN55BE)
//     Drive/Inputs/In/nDataIn1 <-> Transmit PDO mapping 1/Following error actual value
//     Drive/Inputs/In/nDataIn3[0] <-> Transmit PDO mapping 1/Torque actual value
//     Drive/Inputs/In/nDcOutputTime <-> InfoData/DcOutputShift
//     Drive/Inputs/In/nState1 <-> Transmit PDO mapping 1/Statusword
//     Drive/Inputs/In/nState2 <-> Transmit PDO mapping 1/Statusword @bit 8
//     Drive/Inputs/In/nState4 @bit 1 <-> WcState/InputToggle
//     Drive/Inputs/In/nState4 <-> WcState/WcState
//     Drive/Inputs/In/nState5 <-> Transmit PDO mapping 1/Modes of operation display
//     Drive/Outputs/Out/nCtrl1 <-> Receive PDO mapping 1/Controlword
//     Drive/Outputs/Out/nCtrl2 <-> Receive PDO mapping 1/Controlword @bit 8
//     Drive/Outputs/Out/nCtrl5 <-> Receive PDO mapping 1/Modes of operation
//     Drive/Outputs/Out/nDataOut1 <-> Receive PDO mapping 1/Target position
//     Enc/Inputs/In/nDataIn1 <-> Transmit PDO mapping 1/Position actual value
//     Enc/Inputs/In/nDataIn3 <-> Transmit PDO mapping 1/Touch probe pos1 pos value
//     Enc/Inputs/In/nDcInputTime <-> InfoData/DcInputShift
//     Enc/Inputs/In/nState4 @bit 1 <-> WcState/InputToggle
//     Enc/Inputs/In/nState4 <-> WcState/WcState
//     Enc/Inputs/In/nState5 <-> Transmit PDO mapping 1/Touch probe status
//     Enc/Inputs/In/nState6 <-> Transmit PDO mapping 1/Touch probe status @bit 8
//     Enc/Outputs/Out/nCtrl5 <-> Receive PDO mapping 1/Touch probe function
//     Enc/Outputs/Out/nCtrl6 <-> Receive PDO mapping 1/Touch probe function @bit 8
//   NC-Task 1 SAF/Axes/Axis5_RightArm_Left <-> Device 4 (EtherCAT)/Drive RightArm Left (MDDLN55BE)
//     Drive/Inputs/In/nDataIn1 <-> Transmit PDO mapping 1/Following error actual value
//     Drive/Inputs/In/nDataIn3[0] <-> Transmit PDO mapping 1/Torque actual value
//     Drive/Inputs/In/nDcOutputTime <-> InfoData/DcOutputShift
//     Drive/Inputs/In/nState1 <-> Transmit PDO mapping 1/Statusword
//     Drive/Inputs/In/nState2 <-> Transmit PDO mapping 1/Statusword @bit 8
//     Drive/Inputs/In/nState4 @bit 1 <-> WcState/InputToggle
//     Drive/Inputs/In/nState4 <-> WcState/WcState
//     Drive/Inputs/In/nState5 <-> Transmit PDO mapping 1/Modes of operation display
//     Drive/Outputs/Out/nCtrl1 <-> Receive PDO mapping 1/Controlword
//     Drive/Outputs/Out/nCtrl2 <-> Receive PDO mapping 1/Controlword @bit 8
//     Drive/Outputs/Out/nCtrl5 <-> Receive PDO mapping 1/Modes of operation
//     Drive/Outputs/Out/nDataOut1 <-> Receive PDO mapping 1/Target position
//     Enc/Inputs/In/nDataIn1 <-> Transmit PDO mapping 1/Position actual value
//     Enc/Inputs/In/nDataIn3 <-> Transmit PDO mapping 1/Touch probe pos1 pos value
//     Enc/Inputs/In/nDcInputTime <-> InfoData/DcInputShift
//     Enc/Inputs/In/nState4 @bit 1 <-> WcState/InputToggle
//     Enc/Inputs/In/nState4 <-> WcState/WcState
//     Enc/Inputs/In/nState5 <-> Transmit PDO mapping 1/Touch probe status
//     Enc/Inputs/In/nState6 <-> Transmit PDO mapping 1/Touch probe status @bit 8
//     Enc/Outputs/Out/nCtrl5 <-> Receive PDO mapping 1/Touch probe function
//     Enc/Outputs/Out/nCtrl6 <-> Receive PDO mapping 1/Touch probe function @bit 8
//   NC-Task 1 SAF/Axes/Axis6_RightArm_Right <-> Device 4 (EtherCAT)/Drive RightArm Right (MDDLN55BE)
//     Drive/Inputs/In/nDataIn1 <-> Transmit PDO mapping 1/Following error actual value
//     Drive/Inputs/In/nDataIn3[0] <-> Transmit PDO mapping 1/Torque actual value
//     Drive/Inputs/In/nDcOutputTime <-> InfoData/DcOutputShift
//     Drive/Inputs/In/nState1 <-> Transmit PDO mapping 1/Statusword
//     Drive/Inputs/In/nState2 <-> Transmit PDO mapping 1/Statusword @bit 8
//     Drive/Inputs/In/nState4 @bit 1 <-> WcState/InputToggle
//     Drive/Inputs/In/nState4 <-> WcState/WcState
//     Drive/Inputs/In/nState5 <-> Transmit PDO mapping 1/Modes of operation display
//     Drive/Outputs/Out/nCtrl1 <-> Receive PDO mapping 1/Controlword
//     Drive/Outputs/Out/nCtrl2 <-> Receive PDO mapping 1/Controlword @bit 8
//     Drive/Outputs/Out/nCtrl5 <-> Receive PDO mapping 1/Modes of operation
//     Drive/Outputs/Out/nDataOut1 <-> Receive PDO mapping 1/Target position
//     Enc/Inputs/In/nDataIn1 <-> Transmit PDO mapping 1/Position actual value
//     Enc/Inputs/In/nDataIn3 <-> Transmit PDO mapping 1/Touch probe pos1 pos value
//     Enc/Inputs/In/nDcInputTime <-> InfoData/DcInputShift
//     Enc/Inputs/In/nState4 @bit 1 <-> WcState/InputToggle
//     Enc/Inputs/In/nState4 <-> WcState/WcState
//     Enc/Inputs/In/nState5 <-> Transmit PDO mapping 1/Touch probe status
//     Enc/Inputs/In/nState6 <-> Transmit PDO mapping 1/Touch probe status @bit 8
//     Enc/Outputs/Out/nCtrl5 <-> Receive PDO mapping 1/Touch probe function
//     Enc/Outputs/Out/nCtrl6 <-> Receive PDO mapping 1/Touch probe function @bit 8
//   NC-Task 1 SAF/Axes/Axis7_RightArm_Wrist <-> Device 4 (EtherCAT)/Drive RightArm Wrist (MBDLN25BE)
//     Drive/Inputs/In/nDataIn1 <-> Transmit PDO mapping 1/Following error actual value
//     Drive/Inputs/In/nDataIn3[0] <-> Transmit PDO mapping 1/Torque actual value
//     Drive/Inputs/In/nDcOutputTime <-> InfoData/DcOutputShift
//     Drive/Inputs/In/nState1 <-> Transmit PDO mapping 1/Statusword
//     Drive/Inputs/In/nState2 <-> Transmit PDO mapping 1/Statusword @bit 8
//     Drive/Inputs/In/nState4 @bit 1 <-> WcState/InputToggle
//     Drive/Inputs/In/nState4 <-> WcState/WcState
//     Drive/Inputs/In/nState5 <-> Transmit PDO mapping 1/Modes of operation display
//     Drive/Outputs/Out/nCtrl1 <-> Receive PDO mapping 1/Controlword
//     Drive/Outputs/Out/nCtrl2 <-> Receive PDO mapping 1/Controlword @bit 8
//     Drive/Outputs/Out/nCtrl5 <-> Receive PDO mapping 1/Modes of operation
//     Drive/Outputs/Out/nDataOut1 <-> Receive PDO mapping 1/Target position
//     Enc/Inputs/In/nDataIn1 <-> Transmit PDO mapping 1/Position actual value
//     Enc/Inputs/In/nDataIn3 <-> Transmit PDO mapping 1/Touch probe pos1 pos value
//     Enc/Inputs/In/nDcInputTime <-> InfoData/DcInputShift
//     Enc/Inputs/In/nState4 @bit 1 <-> WcState/InputToggle
//     Enc/Inputs/In/nState4 <-> WcState/WcState
//     Enc/Inputs/In/nState5 <-> Transmit PDO mapping 1/Touch probe status
//     Enc/Inputs/In/nState6 <-> Transmit PDO mapping 1/Touch probe status @bit 8
//     Enc/Outputs/Out/nCtrl5 <-> Receive PDO mapping 1/Touch probe function
//     Enc/Outputs/Out/nCtrl6 <-> Receive PDO mapping 1/Touch probe function @bit 8
//   NC-Task 1 SAF/Axes/Axis8_RightArm_Lift <-> Device 4 (EtherCAT)/Drive RightArm Lift (MDDLN55BE)
//     Drive/Inputs/In/nDataIn1 <-> Transmit PDO mapping 1/Following error actual value
//     Drive/Inputs/In/nDataIn3[0] <-> Transmit PDO mapping 1/Torque actual value
//     Drive/Inputs/In/nDcOutputTime <-> InfoData/DcOutputShift
//     Drive/Inputs/In/nState1 <-> Transmit PDO mapping 1/Statusword
//     Drive/Inputs/In/nState2 <-> Transmit PDO mapping 1/Statusword @bit 8
//     Drive/Inputs/In/nState4 @bit 1 <-> WcState/InputToggle
//     Drive/Inputs/In/nState4 <-> WcState/WcState
//     Drive/Inputs/In/nState5 <-> Transmit PDO mapping 1/Modes of operation display
//     Drive/Outputs/Out/nCtrl1 <-> Receive PDO mapping 1/Controlword
//     Drive/Outputs/Out/nCtrl2 <-> Receive PDO mapping 1/Controlword @bit 8
//     Drive/Outputs/Out/nCtrl5 <-> Receive PDO mapping 1/Modes of operation
//     Drive/Outputs/Out/nDataOut1 <-> Receive PDO mapping 1/Target position
//     Enc/Inputs/In/nDataIn1 <-> Transmit PDO mapping 1/Position actual value
//     Enc/Inputs/In/nDataIn3 <-> Transmit PDO mapping 1/Touch probe pos1 pos value
//     Enc/Inputs/In/nDcInputTime <-> InfoData/DcInputShift
//     Enc/Inputs/In/nState4 @bit 1 <-> WcState/InputToggle
//     Enc/Inputs/In/nState4 <-> WcState/WcState
//     Enc/Inputs/In/nState5 <-> Transmit PDO mapping 1/Touch probe status
//     Enc/Inputs/In/nState6 <-> Transmit PDO mapping 1/Touch probe status @bit 8
//     Enc/Outputs/Out/nCtrl5 <-> Receive PDO mapping 1/Touch probe function
//     Enc/Outputs/Out/nCtrl6 <-> Receive PDO mapping 1/Touch probe function @bit 8
//   NC-Task 1 SAF/Axes/Axis9_BigGate_Left <-> Device 4 (EtherCAT)/Drive BigGate Left (MDDLN55BE)
//     Drive/Inputs/In/nDataIn1 <-> Transmit PDO mapping 1/Following error actual value
//     Drive/Inputs/In/nDataIn3[0] <-> Transmit PDO mapping 1/Torque actual value
//     Drive/Inputs/In/nDcOutputTime <-> InfoData/DcOutputShift
//     Drive/Inputs/In/nState1 <-> Transmit PDO mapping 1/Statusword
//     Drive/Inputs/In/nState2 <-> Transmit PDO mapping 1/Statusword @bit 8
//     Drive/Inputs/In/nState4 @bit 1 <-> WcState/InputToggle
//     Drive/Inputs/In/nState4 <-> WcState/WcState
//     Drive/Inputs/In/nState5 <-> Transmit PDO mapping 1/Modes of operation display
//     Drive/Outputs/Out/nCtrl1 <-> Receive PDO mapping 1/Controlword
//     Drive/Outputs/Out/nCtrl2 <-> Receive PDO mapping 1/Controlword @bit 8
//     Drive/Outputs/Out/nCtrl5 <-> Receive PDO mapping 1/Modes of operation
//     Drive/Outputs/Out/nDataOut1 <-> Receive PDO mapping 1/Target position
//     Enc/Inputs/In/nDataIn1 <-> Transmit PDO mapping 1/Position actual value
//     Enc/Inputs/In/nDataIn3 <-> Transmit PDO mapping 1/Touch probe pos1 pos value
//     Enc/Inputs/In/nDcInputTime <-> InfoData/DcInputShift
//     Enc/Inputs/In/nState4 @bit 1 <-> WcState/InputToggle
//     Enc/Inputs/In/nState4 <-> WcState/WcState
//     Enc/Inputs/In/nState5 <-> Transmit PDO mapping 1/Touch probe status
//     Enc/Inputs/In/nState6 <-> Transmit PDO mapping 1/Touch probe status @bit 8
//     Enc/Outputs/Out/nCtrl5 <-> Receive PDO mapping 1/Touch probe function
//     Enc/Outputs/Out/nCtrl6 <-> Receive PDO mapping 1/Touch probe function @bit 8
//   UnloadRobot/UnloadRobot Instance <-> Device 3 (EtherCAT)/Drive LeftWheel Steer (XMC_ESC)
//     PlcTask Outputs/WheelControl.WheelDriver_ModesOfOperation <-> RxPDO/Modes of operation
//   UnloadRobot/UnloadRobot Instance <-> Device 3 (EtherCAT)/Drive LeftWheel Walk (XMC_ESC)
//     PlcTask Outputs/WheelControl.WheelDriver_ModesOfOperation <-> RxPDO/Modes of operation
//   UnloadRobot/UnloadRobot Instance <-> Device 3 (EtherCAT)/Drive RightWheel Steer (XMC_ESC)
//     PlcTask Outputs/WheelControl.WheelDriver_ModesOfOperation <-> RxPDO/Modes of operation
//   UnloadRobot/UnloadRobot Instance <-> Device 3 (EtherCAT)/Drive RightWheel Walk (XMC_ESC)
//     PlcTask Outputs/WheelControl.WheelDriver_ModesOfOperation <-> RxPDO/Modes of operation
//   UnloadRobot/UnloadRobot Instance <-> Device 3 (EtherCAT)/Term 8 (EK1200)/Term 17 (EL1809)
//     PlcTask Inputs/Robot_Control_State.bEmergencyStopBtn <-> Channel 3/Input
//     PlcTask Inputs/Robot_Control_State.bGreenBtn <-> Channel 4/Input
//     PlcTask Inputs/Robot_Control_State.bRedBtn <-> Channel 6/Input
//     PlcTask Inputs/Robot_Control_State.bRemoteCtrl_1btn <-> Channel 14/Input
//     PlcTask Inputs/Robot_Control_State.bRemoteCtrl_2btn <-> Channel 15/Input
//     PlcTask Inputs/Robot_Control_State.bRemoteCtrl_Down <-> Channel 9/Input
//     PlcTask Inputs/Robot_Control_State.bRemoteCtrl_East <-> Channel 10/Input
//     PlcTask Inputs/Robot_Control_State.bRemoteCtrl_North <-> Channel 13/Input
//     PlcTask Inputs/Robot_Control_State.bRemoteCtrl_Online <-> Channel 7/Input
//     PlcTask Inputs/Robot_Control_State.bRemoteCtrl_South <-> Channel 12/Input
//     PlcTask Inputs/Robot_Control_State.bRemoteCtrl_Up <-> Channel 8/Input
//     PlcTask Inputs/Robot_Control_State.bRemoteCtrl_West <-> Channel 11/Input
//     PlcTask Inputs/Robot_Control_State.bTeachBoxAuto <-> Channel 2/Input
//     PlcTask Inputs/Robot_Control_State.bTeachBoxRemote <-> Channel 1/Input
//     PlcTask Inputs/Robot_Control_State.bYellowBtn <-> Channel 5/Input
//     PlcTask Inputs/Robot_Control_State.b_BackBeltCtrlBoxWarning <-> Channel 16/Input
//   UnloadRobot/UnloadRobot Instance <-> Device 3 (EtherCAT)/Term 8 (EK1200)/Term 18 (EL1809)
//     PlcTask Inputs/Robot_Control_State.bLeftArm_Sucker{1..8}_Completed <-> Channel {1..8}/Input  (8 links)
//     PlcTask Inputs/Robot_Control_State.bRightArm_Sucker{1..8}_Completed <-> Channel {9..16}/Input  (8 links)
//   UnloadRobot/UnloadRobot Instance <-> Device 3 (EtherCAT)/Term 8 (EK1200)/Term 19 (EL1809)
//     PlcTask Inputs/Robot_Control_State.bCrash_Sensor_Back <-> Channel 2/Input
//     PlcTask Inputs/Robot_Control_State.bCrash_Sensor_Front <-> Channel 1/Input
//     PlcTask Inputs/Robot_Control_State.bPumpPhaseSequenceProtectionOK <-> Channel 9/Input
//   UnloadRobot/UnloadRobot Instance <-> Device 3 (EtherCAT)/Term 8 (EK1200)/Term 20 (EL2809)
//     PlcTask Outputs/Robot_Control_State.bAxis_GunTong_Back <-> Channel 10/Output
//     PlcTask Outputs/Robot_Control_State.bAxis_GunTong_Left <-> Channel 11/Output
//     PlcTask Outputs/Robot_Control_State.bAxis_GunTong_Middle <-> Channel 13/Output
//     PlcTask Outputs/Robot_Control_State.bAxis_GunTong_Right <-> Channel 12/Output
//     PlcTask Outputs/Robot_Control_State.bBtnLed_Green_Enable <-> Channel 4/Output
//     PlcTask Outputs/Robot_Control_State.bBtnLed_Red_Enable <-> Channel 6/Output
//     PlcTask Outputs/Robot_Control_State.bBtnLed_Yellow_Enable <-> Channel 5/Output
//     PlcTask Outputs/Robot_Control_State.bFrontLight_Left_Enable <-> Channel 7/Output
//     PlcTask Outputs/Robot_Control_State.bFrontLight_Right_Enable <-> Channel 8/Output
//     PlcTask Outputs/Robot_Control_State.bPumpMotor_Enable <-> Channel 9/Output
//     PlcTask Outputs/Robot_Control_State.bTriColorLed_Green_Enable <-> Channel 1/Output
//     PlcTask Outputs/Robot_Control_State.bTriColorLed_Red_Enable <-> Channel 3/Output
//     PlcTask Outputs/Robot_Control_State.bTriColorLed_Yellow_Enable <-> Channel 2/Output
//   UnloadRobot/UnloadRobot Instance <-> Device 3 (EtherCAT)/Term 8 (EK1200)/Term 21 (EL2809)
//     PlcTask Outputs/Robot_Control_State.bLeftArm_SV{1..8} <-> Channel {1..8}/Output  (8 links)
//     PlcTask Outputs/Robot_Control_State.bRightArm_SV{1..8} <-> Channel {9..16}/Output  (8 links)
//   UnloadRobot/UnloadRobot Instance <-> Device 4 (EtherCAT)/Drive BackGate Left (MCDLN35BE)
//     PlcTask Inputs/Robot_Motor.axis_BackGate_Left_Torque <-> Transmit PDO mapping 1/Torque actual value
//   UnloadRobot/UnloadRobot Instance <-> Device 4 (EtherCAT)/Drive BackGate Right(MCDLN35BE)
//     PlcTask Inputs/Robot_Motor.axis_BackGate_Right_Torque <-> Transmit PDO mapping 1/Torque actual value
//   UnloadRobot/UnloadRobot Instance <-> Device 4 (EtherCAT)/Drive BigGate Left (MDDLN55BE)
//     PlcTask Inputs/Robot_Motor.axis_BigGate_Left_Torque <-> Transmit PDO mapping 1/Torque actual value
//   UnloadRobot/UnloadRobot Instance <-> Device 4 (EtherCAT)/Drive BigGate Right (MDDLN55BE)
//     PlcTask Inputs/Robot_Motor.axis_BigGate_Right_Torque <-> Transmit PDO mapping 1/Torque actual value
//   UnloadRobot/UnloadRobot Instance <-> Device 4 (EtherCAT)/Drive LeftArm Left (MDDLN55BE)
//     PlcTask Inputs/Robot_Motor.axis_LeftArm_Left_Torque <-> Transmit PDO mapping 1/Torque actual value
//   UnloadRobot/UnloadRobot Instance <-> Device 4 (EtherCAT)/Drive LeftArm Lift (MDDLN55BE)
//     PlcTask Inputs/Robot_Motor.axis_LeftArm_Lift_Torque <-> Transmit PDO mapping 1/Torque actual value
//   UnloadRobot/UnloadRobot Instance <-> Device 4 (EtherCAT)/Drive LeftArm Right (MDDLN55BE)
//     PlcTask Inputs/Robot_Motor.axis_LeftArm_Right_Torque <-> Transmit PDO mapping 1/Torque actual value
//   UnloadRobot/UnloadRobot Instance <-> Device 4 (EtherCAT)/Drive LeftArm Wrist (MBDLN25BE)
//     PlcTask Inputs/Robot_Motor.axis_LeftArm_Wrist_Torque <-> Transmit PDO mapping 1/Torque actual value
//   UnloadRobot/UnloadRobot Instance <-> Device 4 (EtherCAT)/Drive RightArm Left (MDDLN55BE)
//     PlcTask Inputs/Robot_Motor.axis_RightArm_Left_Torque <-> Transmit PDO mapping 1/Torque actual value
//   UnloadRobot/UnloadRobot Instance <-> Device 4 (EtherCAT)/Drive RightArm Lift (MDDLN55BE)
//     PlcTask Inputs/Robot_Motor.axis_RightArm_Lift_Torque <-> Transmit PDO mapping 1/Torque actual value
//   UnloadRobot/UnloadRobot Instance <-> Device 4 (EtherCAT)/Drive RightArm Right (MDDLN55BE)
//     PlcTask Inputs/Robot_Motor.axis_RightArm_Right_Torque <-> Transmit PDO mapping 1/Torque actual value
//   UnloadRobot/UnloadRobot Instance <-> Device 4 (EtherCAT)/Drive RightArm Wrist (MBDLN25BE)
//     PlcTask Inputs/Robot_Motor.axis_RightArm_Wrist_Torque <-> Transmit PDO mapping 1/Torque actual value
//   UnloadRobot/UnloadRobot Instance <-> Device 4 (EtherCAT)/Drive SmallGate Left (MDDLN45BE)
//     PlcTask Inputs/Robot_Motor.axis_SmallGate_Left_Torque <-> Transmit PDO mapping 1/Torque actual value
//   UnloadRobot/UnloadRobot Instance <-> Device 4 (EtherCAT)/Drive SmallGate Right (MDDLN45BE)
//     PlcTask Inputs/Robot_Motor.axis_SmallGate_Right_Torque <-> Transmit PDO mapping 1/Torque actual value
//   UnloadRobot/UnloadRobot Instance <-> Device 5 (COM Port)
//     PlcTask Inputs/GVL_SerialComunication.pComIn/D[{0..63}] <-> Inputs/Data{1..64}  (64 links)
//     PlcTask Inputs/GVL_SerialComunication.pComIn/SerStatus <-> Inputs/Status
//     PlcTask Outputs/GVL_SerialComunication.pComOut/D[{0..63}] <-> Outputs/Data{1..64}  (64 links)
//     PlcTask Outputs/GVL_SerialComunication.pComOut/SerCtrl <-> Outputs/Ctrl
//   UnloadRobot/UnloadRobot Instance <-> NC-Task 1 SAF/Axes/Axis10_BigGate_Right
//     PlcTask Inputs/Robot_Motor.axis_BigGate_Right.NcToPlc <-> Outputs/ToPlc
//     PlcTask Inputs/Robot_Status_Info.bDriverDeviceErrorCode_axis_BigGate_Right <-> Outputs/ToPlc/ErrorCode
//     PlcTask Inputs/Robot_Status_Info.bDriverDeviceError_axis_BigGate_Right <-> Outputs/ToPlc/StateDWord/DriveDeviceError
//     PlcTask Outputs/Robot_Motor.axis_BigGate_Right.PlcToNc <-> Inputs/FromPlc
//   UnloadRobot/UnloadRobot Instance <-> NC-Task 1 SAF/Axes/Axis11_SmallGate_Left
//     PlcTask Inputs/Robot_Motor.axis_SmallGate_Left.NcToPlc <-> Outputs/ToPlc
//     PlcTask Inputs/Robot_Status_Info.bDriverDeviceErrorCode_axis_SmallGate_Left <-> Outputs/ToPlc/ErrorCode
//     PlcTask Inputs/Robot_Status_Info.bDriverDeviceError_axis_SmallGate_Left <-> Outputs/ToPlc/StateDWord/DriveDeviceError
//     PlcTask Outputs/Robot_Motor.axis_SmallGate_Left.PlcToNc <-> Inputs/FromPlc
//   UnloadRobot/UnloadRobot Instance <-> NC-Task 1 SAF/Axes/Axis12_SmallGate_Right
//     PlcTask Inputs/Robot_Motor.axis_SmallGate_Right.NcToPlc <-> Outputs/ToPlc
//     PlcTask Inputs/Robot_Status_Info.bDriverDeviceErrorCode_axis_SmallGate_Right <-> Outputs/ToPlc/ErrorCode
//     PlcTask Inputs/Robot_Status_Info.bDriverDeviceError_axis_SmallGate_Right <-> Outputs/ToPlc/StateDWord/DriveDeviceError
//     PlcTask Outputs/Robot_Motor.axis_SmallGate_Right.PlcToNc <-> Inputs/FromPlc
//   UnloadRobot/UnloadRobot Instance <-> NC-Task 1 SAF/Axes/Axis13_BackGate_Left
//     PlcTask Inputs/Robot_Motor.axis_BackGate_Left.NcToPlc <-> Outputs/ToPlc
//     PlcTask Inputs/Robot_Status_Info.bDriverDeviceErrorCode_axis_BackGate_Left <-> Outputs/ToPlc/ErrorCode
//     PlcTask Inputs/Robot_Status_Info.bDriverDeviceError_axis_BackGate_Left <-> Outputs/ToPlc/StateDWord/DriveDeviceError
//     PlcTask Outputs/Robot_Motor.axis_BackGate_Left.PlcToNc <-> Inputs/FromPlc
//   UnloadRobot/UnloadRobot Instance <-> NC-Task 1 SAF/Axes/Axis14_BackGate_Right
//     PlcTask Inputs/Robot_Motor.axis_BackGate_Right.NcToPlc <-> Outputs/ToPlc
//     PlcTask Inputs/Robot_Status_Info.bDriverDeviceErrorCode_axis_BackGate_Right <-> Outputs/ToPlc/ErrorCode
//     PlcTask Inputs/Robot_Status_Info.bDriverDeviceError_axis_BackGate_Right <-> Outputs/ToPlc/StateDWord/DriveDeviceError
//     PlcTask Outputs/Robot_Motor.axis_BackGate_Right.PlcToNc <-> Inputs/FromPlc
//   UnloadRobot/UnloadRobot Instance <-> NC-Task 1 SAF/Axes/Axis15_RightWheel_Steer
//     PlcTask Inputs/Robot_Motor.axis_RightWheel_Steer.NcToPlc <-> Outputs/ToPlc
//     PlcTask Inputs/Robot_Status_Info.bDriverDeviceErrorCode_axis_RightWheel_Steer <-> Outputs/ToPlc/ErrorCode
//     PlcTask Inputs/Robot_Status_Info.bDriverDeviceError_axis_RightWheel_Steer <-> Outputs/ToPlc/StateDWord/DriveDeviceError
//     PlcTask Outputs/Robot_Motor.axis_RightWheel_Steer.PlcToNc <-> Inputs/FromPlc
//   UnloadRobot/UnloadRobot Instance <-> NC-Task 1 SAF/Axes/Axis16_RightWheel_Walk
//     PlcTask Inputs/Robot_Motor.axis_RightWheel_Walk.NcToPlc <-> Outputs/ToPlc
//     PlcTask Inputs/Robot_Status_Info.bDriverDeviceErrorCode_axis_RightWheel_Walk <-> Outputs/ToPlc/ErrorCode
//     PlcTask Inputs/Robot_Status_Info.bDriverDeviceError_axis_RightWheel_Walk <-> Outputs/ToPlc/StateDWord/DriveDeviceError
//     PlcTask Outputs/Robot_Motor.axis_RightWheel_Walk.PlcToNc <-> Inputs/FromPlc
//   UnloadRobot/UnloadRobot Instance <-> NC-Task 1 SAF/Axes/Axis17_LeftWheel_Steer
//     PlcTask Inputs/Robot_Motor.axis_LeftWheel_Steer.NcToPlc <-> Outputs/ToPlc
//     PlcTask Inputs/Robot_Status_Info.bDriverDeviceErrorCode_axis_LeftWheel_Steer <-> Outputs/ToPlc/ErrorCode
//     PlcTask Inputs/Robot_Status_Info.bDriverDeviceError_axis_LeftWheel_Steer <-> Outputs/ToPlc/StateDWord/DriveDeviceError
//     PlcTask Outputs/Robot_Motor.axis_LeftWheel_Steer.PlcToNc <-> Inputs/FromPlc
//   UnloadRobot/UnloadRobot Instance <-> NC-Task 1 SAF/Axes/Axis18_LeftWheel_Walk
//     PlcTask Inputs/Robot_Motor.axis_LeftWheel_Walk.NcToPlc <-> Outputs/ToPlc
//     PlcTask Inputs/Robot_Status_Info.bDriverDeviceErrorCode_axis_LeftWheel_Walk <-> Outputs/ToPlc/ErrorCode
//     PlcTask Inputs/Robot_Status_Info.bDriverDeviceError_axis_LeftWheel_Walk <-> Outputs/ToPlc/StateDWord/DriveDeviceError
//     PlcTask Outputs/Robot_Motor.axis_LeftWheel_Walk.PlcToNc <-> Inputs/FromPlc
//   UnloadRobot/UnloadRobot Instance <-> NC-Task 1 SAF/Axes/Axis1_LeftArm_Left
//     PlcTask Inputs/Robot_Motor.axis_LeftArm_Left.NcToPlc <-> Outputs/ToPlc
//     PlcTask Inputs/Robot_Status_Info.bDriverDeviceErrorCode_axis_LeftArm_Left <-> Outputs/ToPlc/ErrorCode
//     PlcTask Inputs/Robot_Status_Info.bDriverDeviceError_axis_LeftArm_Left <-> Outputs/ToPlc/StateDWord/DriveDeviceError
//     PlcTask Outputs/Robot_Motor.axis_LeftArm_Left.PlcToNc <-> Inputs/FromPlc
//   UnloadRobot/UnloadRobot Instance <-> NC-Task 1 SAF/Axes/Axis2_LeftArm_Right
//     PlcTask Inputs/Robot_Motor.axis_LeftArm_Right.NcToPlc <-> Outputs/ToPlc
//     PlcTask Inputs/Robot_Status_Info.bDriverDeviceErrorCode_axis_LeftArm_Right <-> Outputs/ToPlc/ErrorCode
//     PlcTask Inputs/Robot_Status_Info.bDriverDeviceError_axis_LeftArm_Right <-> Outputs/ToPlc/StateDWord/DriveDeviceError
//     PlcTask Outputs/Robot_Motor.axis_LeftArm_Right.PlcToNc <-> Inputs/FromPlc
//   UnloadRobot/UnloadRobot Instance <-> NC-Task 1 SAF/Axes/Axis3_LeftArm_Wrist
//     PlcTask Inputs/Robot_Motor.axis_LeftArm_Wrist.NcToPlc <-> Outputs/ToPlc
//     PlcTask Inputs/Robot_Status_Info.bDriverDeviceErrorCode_axis_LeftArm_Wrist <-> Outputs/ToPlc/ErrorCode
//     PlcTask Inputs/Robot_Status_Info.bDriverDeviceError_axis_LeftArm_Wrist <-> Outputs/ToPlc/StateDWord/DriveDeviceError
//     PlcTask Outputs/Robot_Motor.axis_LeftArm_Wrist.PlcToNc <-> Inputs/FromPlc
//   UnloadRobot/UnloadRobot Instance <-> NC-Task 1 SAF/Axes/Axis4_LeftArm_Lift
//     PlcTask Inputs/Robot_Motor.axis_LeftArm_Lift.NcToPlc <-> Outputs/ToPlc
//     PlcTask Inputs/Robot_Status_Info.bDriverDeviceErrorCode_axis_LeftArm_Lift <-> Outputs/ToPlc/ErrorCode
//     PlcTask Inputs/Robot_Status_Info.bDriverDeviceError_axis_LeftArm_Lift <-> Outputs/ToPlc/StateDWord/DriveDeviceError
//     PlcTask Outputs/Robot_Motor.axis_LeftArm_Lift.PlcToNc <-> Inputs/FromPlc
//   UnloadRobot/UnloadRobot Instance <-> NC-Task 1 SAF/Axes/Axis5_RightArm_Left
//     PlcTask Inputs/Robot_Motor.axis_RightArm_Left.NcToPlc <-> Outputs/ToPlc
//     PlcTask Inputs/Robot_Status_Info.bDriverDeviceErrorCode_axis_RightArm_Left <-> Outputs/ToPlc/ErrorCode
//     PlcTask Inputs/Robot_Status_Info.bDriverDeviceError_axis_RightArm_Left <-> Outputs/ToPlc/StateDWord/DriveDeviceError
//     PlcTask Outputs/Robot_Motor.axis_RightArm_Left.PlcToNc <-> Inputs/FromPlc
//   UnloadRobot/UnloadRobot Instance <-> NC-Task 1 SAF/Axes/Axis6_RightArm_Right
//     PlcTask Inputs/Robot_Motor.axis_RightArm_Right.NcToPlc <-> Outputs/ToPlc
//     PlcTask Inputs/Robot_Status_Info.bDriverDeviceErrorCode_axis_RightArm_Right <-> Outputs/ToPlc/ErrorCode
//     PlcTask Inputs/Robot_Status_Info.bDriverDeviceError_axis_RightArm_Right <-> Outputs/ToPlc/StateDWord/DriveDeviceError
//     PlcTask Outputs/Robot_Motor.axis_RightArm_Right.PlcToNc <-> Inputs/FromPlc
//   UnloadRobot/UnloadRobot Instance <-> NC-Task 1 SAF/Axes/Axis7_RightArm_Wrist
//     PlcTask Inputs/Robot_Motor.axis_RightArm_Wrist.NcToPlc <-> Outputs/ToPlc
//     PlcTask Inputs/Robot_Status_Info.bDriverDeviceErrorCode_axis_RightArm_Wrist <-> Outputs/ToPlc/ErrorCode
//     PlcTask Inputs/Robot_Status_Info.bDriverDeviceError_axis_RightArm_Wrist <-> Outputs/ToPlc/StateDWord/DriveDeviceError
//     PlcTask Outputs/Robot_Motor.axis_RightArm_Wrist.PlcToNc <-> Inputs/FromPlc
//   UnloadRobot/UnloadRobot Instance <-> NC-Task 1 SAF/Axes/Axis8_RightArm_Lift
//     PlcTask Inputs/Robot_Motor.axis_RightArm_Lift.NcToPlc <-> Outputs/ToPlc
//     PlcTask Inputs/Robot_Status_Info.bDriverDeviceErrorCode_axis_RightArm_Lift <-> Outputs/ToPlc/ErrorCode
//     PlcTask Inputs/Robot_Status_Info.bDriverDeviceError_axis_RightArm_Lift <-> Outputs/ToPlc/StateDWord/DriveDeviceError
//     PlcTask Outputs/Robot_Motor.axis_RightArm_Lift.PlcToNc <-> Inputs/FromPlc
//   UnloadRobot/UnloadRobot Instance <-> NC-Task 1 SAF/Axes/Axis9_BigGate_Left
//     PlcTask Inputs/Robot_Motor.axis_BigGate_Left.NcToPlc <-> Outputs/ToPlc
//     PlcTask Inputs/Robot_Status_Info.bDriverDeviceErrorCode_axis_BigGate_Left <-> Outputs/ToPlc/ErrorCode
//     PlcTask Inputs/Robot_Status_Info.bDriverDeviceError_axis_BigGate_Left <-> Outputs/ToPlc/StateDWord/DriveDeviceError
//     PlcTask Outputs/Robot_Motor.axis_BigGate_Left.PlcToNc <-> Inputs/FromPlc

CONFIGURATION UnloadRobot
    RESOURCE PLC ON TwinCAT3
        TASK PlcTask(INTERVAL := T#10ms, PRIORITY := 20);
        PROGRAM AxisAbs WITH PlcTask : AxisAbs;
        PROGRAM AxisAllCtrl WITH PlcTask : AxisAllCtrl;
        PROGRAM AxisJog WITH PlcTask : AxisJog;
        PROGRAM AxisPowerOn WITH PlcTask : AxisPowerOn;
        PROGRAM AxisReset WITH PlcTask : AxisReset;
        PROGRAM AxisStop WITH PlcTask : AxisStop;
        PROGRAM GateMove WITH PlcTask : GateMove;
        PROGRAM LeftArmManualCtrlMove WITH PlcTask : LeftArmManualCtrlMove;
        PROGRAM MAIN WITH PlcTask : MAIN;
        PROGRAM MoveExtPos WITH PlcTask : MoveExtPos;
        PROGRAM RightArmManualCtrlMove WITH PlcTask : RightArmManualCtrlMove;
        PROGRAM WheelControl WITH PlcTask : WheelControl;
        PROGRAM TBoxCtrl WITH PlcTask : TBoxCtrl;
    END_RESOURCE
END_CONFIGURATION

// ---- DUTs/Angles.TcDUT
TYPE Angles :
STRUCT
	theta1_right	:LREAL;
	theta2_left		:LREAL;
END_STRUCT
END_TYPE

// ---- DUTs/Box.TcDUT
TYPE Box :
STRUCT
	x				:REAL;
	y				:REAL;
	w				:REAL;
	h				:REAL;
	confidence		:REAL;
	row_index		:REAL;
	part			:REAL;
END_STRUCT
END_TYPE

// ---- DUTs/DUT.TcDUT
TYPE DUT :
UNION
END_UNION
END_TYPE

// ---- DUTs/Points.TcDUT
TYPE Points :
STRUCT
	x:LREAL;
	y:LREAL;
	
END_STRUCT
END_TYPE

// ---- DUTs/SystemStatus.TcDUT
{attribute 'qualified_only'}
{attribute 'strict'}
TYPE SystemStatus :
(
	System_OK := 0,
	ChassisManual_Slow,
	ChassisManual_Fast,
	EmergencyStop:=255
);
END_TYPE

// ---- GVLs/GVL_SerialComunication.TcGVL
//{attribute 'qualified_only'}
VAR_GLOBAL
	//背景通信模块
	BMSSerialCtrl										:SerialLineControl;
	pComIn						AT %I*					:PcComInData;
	pComOut						AT %Q*					:PcComOutData;
	TxBuffer											:combuffer;
	RxBuffer											:combuffer;
	
	//查询命令
	queryBmsStatusCmd			:ARRAY[1..7] OF BYTE	:=[16#DD, 16#A5, 16#03, 16#00, 16#FF, 16#FD, 16#77];
	queryBmsStatusCmdLen		:INT					:=7;
	
END_VAR

// ---- GVLs/Robot_Control_State.TcGVL
//{attribute 'qualified_only'}
VAR_GLOBAL
	
	(*电机操作逆时针为正*)
	
(*======================================== 自定义标志位 Start ======================================*)	
	bManualCtrl_Asm_LeftArm										:BOOL;			// 手动控制标志位-总成-左臂
	bManualCtrl_Asm_RightArm									:BOOL;			// 手动控制标志位-总成-右臂

	bAutoCtrl_Part_LeftWrist									:BOOL;			// 自动控制-单体-腕电机
	bAutoCtrl_Part_RightWrist									:BOOL;			// 自动控制-单体-腕电机	


	// 单轴控制标志位
	bManualCtrl_Part_LeftArm_Left								:BOOL;			
	bManualCtrl_Part_LeftArm_Right								:BOOL;			
	bManualCtrl_Part_LeftArm_Wrist								:BOOL;	
	bManualCtrl_Part_LeftArm_Lift								:BOOL;
	bManualCtrl_Part_RightArm_Left								:BOOL;
	bManualCtrl_Part_RightArm_Right								:BOOL;			
	bManualCtrl_Part_RightArm_Wrist								:BOOL;	
	bManualCtrl_Part_RightArm_Lift								:BOOL;
	bManualCtrl_Part_BigGate_Left								:BOOL;
	bManualCtrl_Part_BigGate_Right								:BOOL;	
	bManualCtrl_Part_SmallGate_Left								:BOOL;
	bManualCtrl_Part_SmallGate_Right							:BOOL;		
	bManualCtrl_Part_BackGate_Left								:BOOL;
	bManualCtrl_Part_BackGate_Right								:BOOL;

	// 合成同步运动标志位		
	bManualCtrl_Asm_BigGate										:BOOL;
	bManualCtrl_Asm_SmallGate									:BOOL;
	bManualCtrl_Asm_BackGate									:BOOL;
	
	
	// 急停激活时大龙门、小龙门、后龙门电子齿轮重新啮合标志位
	// 当Slave轴触发Mc_Stop，会自动取消啮合，需要再次GearIn一下，所以此处设了一个全局变量，恢复急停后统一把三个龙门电子齿轮重新啮合一下。
	bEStopGearInAgain											:BOOL:=TRUE;
	bSmallGate_Gearin_do										:BOOL:=TRUE;
	bBigGate_Gearin_do											:BOOL:=TRUE;
	bBackGate_Gearin_do											:BOOL:=TRUE;

(*======================================== 自定义标志位 End ========================================*)	



(*=================================================    走位置演示    =======================================*)

	bAutoMovePosSet												:BOOL;			// 走位置演示
	
	
(*=================================================    走位置演示    =======================================*)



	

(*========================================电机使能标志位 Start =====================================*)	
	
	// 左臂电机
	bAxis_LeftArm_Wrist_Enable									:BOOL;				//左臂_腕电机使能	
	bAxis_LeftArm_Left_Enable									:BOOL;				//左臂_左电机使能
	bAxis_LeftArm_Right_Enable									:BOOL;				//左臂_右电机使能	
	bAxis_LeftArm_Lift_Enable									:BOOL;				//左臂_升电机使能	

	// 右臂电机
	bAxis_RightArm_Wrist_Enable									:BOOL;				//右臂_腕电机使能	
	bAxis_RightArm_Left_Enable									:BOOL;				//右臂_左电机使能
	bAxis_RightArm_Right_Enable									:BOOL;				//右臂_右电机使能
	bAxis_RightArm_Lift_Enable									:BOOL;				//右臂_升电机使能
	                                                                            	
	// 小龙门电机                                                                    	
	bAxis_SmallGate_Left_Enable									:BOOL;				//小门_左电机使能
	bAxis_SmallGate_Right_Enable								:BOOL;				//小门_右电机使能
                                                                                	
	// 大龙门单电机                                                                   	
	bAxis_BigGate_Left_Enable									:BOOL;				//大门_左电机使能
	bAxis_BigGate_Right_Enable									:BOOL;				//大门_右电机使能
	                                                                            	
	// 后龙门单电机                                                                   	
	bAxis_BackGate_Left_Enable									:BOOL;				//后门_左电机使能
	bAxis_BackGate_Right_Enable									:BOOL;				//后门_右电机使能
	
	// 右轮
	bAxis_RightWheel_Steer_Enable								:BOOL;
	bAxis_RightWheel_Walk_Enable								:BOOL;
	
	// 左轮
	bAxis_LeftWheel_Steer_Enable								:BOOL;
	bAxis_LeftWheel_Walk_Enable									:BOOL;
	
	
	// 所有轴
	bAxis_All_Enable											:BOOL;				//所有电机使能
	bAxis_All_Disable											:BOOL;				//所有电机失能
	
	
	// 所有轴使能标志位的地址交给此Group来管理
	aAxis_All_Enable_Group 										:ARRAY[1..23] OF POINTER TO BOOL:=[
																									ADR(bAxis_LeftArm_Wrist_Enable),	
																									ADR(bAxis_LeftArm_Left_Enable),	
																									ADR(bAxis_LeftArm_Right_Enable),
																									ADR(bAxis_LeftArm_Lift_Enable),
																									ADR(bAxis_RightArm_Wrist_Enable),	
																									ADR(bAxis_RightArm_Left_Enable),	
																									ADR(bAxis_RightArm_Right_Enable),	
																									ADR(bAxis_RightArm_Lift_Enable),
																									ADR(bAxis_SmallGate_Left_Enable),
																									ADR(bAxis_SmallGate_Right_Enable),
																									ADR(bAxis_BigGate_Left_Enable),	
																									ADR(bAxis_BigGate_Right_Enable),
																									ADR(bAxis_BackGate_Left_Enable),	
																									ADR(bAxis_BackGate_Right_Enable),
																									ADR(bAxis_RightWheel_Steer_Enable),	
																									ADR(bAxis_RightWheel_Walk_Enable),	
																									ADR(bAxis_LeftWheel_Steer_Enable),
																									ADR(bAxis_LeftWheel_Walk_Enable)	
																									
																				 				 ];

(*========================================电机使能标志位 End ======================================*)	




(*======================================== 清故障标志位 Start =====================================*)	

	// 左臂电机
	bAxis_LeftArm_Wrist_Reset									:BOOL;				//左臂_腕电机复位	
	bAxis_LeftArm_Left_Reset									:BOOL;				//左臂_左电机复位
	bAxis_LeftArm_Right_Reset									:BOOL;				//左臂_右电机复位	
	bAxis_LeftArm_Lift_Reset									:BOOL;				//左臂_升电机复位	

	// 右臂电机
	bAxis_RightArm_Wrist_Reset									:BOOL;				//右臂_腕电机复位	
	bAxis_RightArm_Left_Reset									:BOOL;				//右臂_左电机复位
	bAxis_RightArm_Right_Reset									:BOOL;				//右臂_右电机复位
	bAxis_RightArm_Lift_Reset									:BOOL;				//右臂_升电机复位
	                                                                            	
	// 小龙门电机                                                                    	
	bAxis_SmallGate_Left_Reset									:BOOL;				//小门_左电机复位
	bAxis_SmallGate_Right_Reset									:BOOL;				//小门_右电机复位
                                                                                	
	// 大龙门单电机                                                                   	
	bAxis_BigGate_Left_Reset									:BOOL;				//大门_左电机复位
	bAxis_BigGate_Right_Reset									:BOOL;				//大门_右电机复位
	                                                                            	
	// 后龙门单电机                                                                   	
	bAxis_BackGate_Left_Reset									:BOOL;				//后门_左电机复位
	bAxis_BackGate_Right_Reset									:BOOL;				//后门_右电机复位
	
	// 右轮
	bAxis_RightWheel_Steer_Reset								:BOOL;
	bAxis_RightWheel_Walk_Reset								:BOOL;
	
	// 左轮
	bAxis_LeftWheel_Steer_Reset								:BOOL;
	bAxis_LeftWheel_Walk_Reset									:BOOL;
	
	
	
	
	
	
	
	// 所有轴
	bAxis_All_Reset												:BOOL;				//所有电机使能

	// 所有轴使能标志位的地址交给此Group来管理
	aAxis_All_Reset_Group 										:ARRAY[1..23] OF POINTER TO BOOL:=[
																									ADR(bAxis_LeftArm_Wrist_Reset),	
																									ADR(bAxis_LeftArm_Left_Reset),	
																									ADR(bAxis_LeftArm_Right_Reset),
																									ADR(bAxis_LeftArm_Lift_Reset),
																									ADR(bAxis_RightArm_Wrist_Reset),	
																									ADR(bAxis_RightArm_Left_Reset),	
																									ADR(bAxis_RightArm_Right_Reset),	
																									ADR(bAxis_RightArm_Lift_Reset),
																									ADR(bAxis_SmallGate_Left_Reset),
																									ADR(bAxis_SmallGate_Right_Reset),
																									ADR(bAxis_BigGate_Left_Reset),	
																									ADR(bAxis_BigGate_Right_Reset),
																									ADR(bAxis_BackGate_Left_Reset),	
																									ADR(bAxis_BackGate_Right_Reset),
																									ADR(bAxis_RightWheel_Steer_Reset),	
																									ADR(bAxis_RightWheel_Walk_Reset),	
																									ADR(bAxis_LeftWheel_Steer_Reset),
																									ADR(bAxis_LeftWheel_Walk_Reset)	
																									
																				 				 ];


(*======================================== 清故障标志位 End ========================================*)	



(*======================================== 单电机调试MoveAbs标志位 End ========================================*)	
	
	// 左臂电机
	bAxis_LeftArm_Wrist_MoveAbs									:BOOL;				//左臂_腕电机MoveAbs标志位	
	bAxis_LeftArm_Left_MoveAbs									:BOOL;				//左臂_左电机MoveAbs标志位
	bAxis_LeftArm_Right_MoveAbs									:BOOL;				//左臂_右电机MoveAbs标志位	
	bAxis_LeftArm_Lift_MoveAbs									:BOOL;				//左臂_升电机MoveAbs标志位	
                                                                                           
	// 右臂电机                                                                                
	bAxis_RightArm_Wrist_MoveAbs								:BOOL;				//右臂_腕电机MoveAbs标志位	
	bAxis_RightArm_Left_MoveAbs									:BOOL;				//右臂_左电机MoveAbs标志位
	bAxis_RightArm_Right_MoveAbs								:BOOL;				//右臂_右电机MoveAbs标志位
	bAxis_RightArm_Lift_MoveAbs									:BOOL;				//右臂_升电机MoveAbs标志位
	                                                                            	       
	// 小龙门电机                                                                    	       
	bAxis_SmallGate_Left_MoveAbs								:BOOL;				//小门_左电机MoveAbs标志位
	bAxis_SmallGate_Right_MoveAbs								:BOOL;				//小门_右电机MoveAbs标志位
                                                                                	        
	// 大龙门单电机                                                                   	        
	bAxis_BigGate_Left_MoveAbs									:BOOL;				//大门_左电机MoveAbs标志位
	bAxis_BigGate_Right_MoveAbs									:BOOL;				//大门_右电机MoveAbs标志位
	                                                                            	       
	// 后龙门单电机                                                                   	       
	bAxis_BackGate_Left_MoveAbs									:BOOL;				//后门_左电机MoveAbs标志位
	bAxis_BackGate_Right_MoveAbs								:BOOL;				//后门_右电机MoveAbs标志位


(*======================================== 单电机调试MoveAbs标志位  End ========================================*)	





(*======================================== 机器人各轴 MC_Stop标志位 Start ==================================*)
	
	// 左臂电机
	bAxis_LeftArm_Wrist_McStop									:BOOL;			//左臂_腕电机MC_Stop标志位	
	bAxis_LeftArm_Left_McStop									:Bool;			//左臂_左电机MC_Stop标志位
	bAxis_LeftArm_Right_McStop									:Bool;			//左臂_右电机MC_Stop标志位
	bAxis_LeftArm_Lift_McStop									:Bool;			//左臂_升电机MC_Stop标志位
	                                                                                        
	// 右臂电机                                                                                 
	bAxis_RightArm_Wrist_McStop									:Bool;			//右臂_腕电机MC_Stop标志位	
	bAxis_RightArm_Left_McStop									:Bool;			//右臂_左电机MC_Stop标志位
	bAxis_RightArm_Right_McStop									:Bool;			//右臂_右电机MC_Stop标志位
	bAxis_RightArm_Lift_McStop									:Bool;			//右臂_升电机MC_Stop标志位
	                                                                                        
	// 小龙门电机                                                                                
	bAxis_SmallGate_Left_McStop									:Bool;			//小门_左电机MC_Stop标志位
	bAxis_SmallGate_Right_McStop								:Bool;			//小门_右电机MC_Stop标志位
	                                                                                        
	// 大龙门单电机                                                                               
	bAxis_BigGate_Left_McStop									:Bool;			//大门_左电机MC_Stop标志位
	bAxis_BigGate_Right_McStop									:Bool;			//大门_右电机MC_Stop标志位
	                                                                                        
	// 后龙门单电机                                                                               
	bAxis_BackGate_Left_McStop									:Bool;			//后门_左电机MC_Stop标志位
	bAxis_BackGate_Right_McStop									:BOOL;			//后门_右电机MC_Stop标志位
	
	// 右轮
	bAxis_RightWheel_Steer_McStop								:BOOL;
	bAxis_RightWheel_Walk_McStop								:BOOL;
	
	// 左轮
	bAxis_LeftWheel_Steer_McStop								:BOOL;
	bAxis_LeftWheel_Walk_McStop									:BOOL;
	
		// 所有轴
	bAxis_All_Stop												:BOOL;			//所有电机使能

	// 所有轴停止标志位的地址交给此Group来管理
	aAxis_All_Stop_Group 										:ARRAY[1..23] OF POINTER TO BOOL:=[
																									ADR(bAxis_LeftArm_Wrist_McStop),	
																									ADR(bAxis_LeftArm_Left_McStop),	
																									ADR(bAxis_LeftArm_Right_McStop),
																									ADR(bAxis_LeftArm_Lift_McStop),
																									ADR(bAxis_RightArm_Wrist_McStop),	
																									ADR(bAxis_RightArm_Left_McStop),	
																									ADR(bAxis_RightArm_Right_McStop),	
																									ADR(bAxis_RightArm_Lift_McStop),
																									ADR(bAxis_SmallGate_Left_McStop),
																									ADR(bAxis_SmallGate_Right_McStop),
																									ADR(bAxis_BigGate_Left_McStop),	
																									ADR(bAxis_BigGate_Right_McStop),
																									ADR(bAxis_BackGate_Left_McStop),	
																									ADR(bAxis_BackGate_Right_McStop),
																									ADR(bAxis_RightWheel_Steer_McStop),
																									ADR(bAxis_RightWheel_Walk_McStop),
																									ADR(bAxis_LeftWheel_Steer_McStop),
																									ADR(bAxis_LeftWheel_Walk_McStop)	
																				 				 ];


(*======================================== 机器人各轴 Mc_Stop标志位 End =====================================*)





	
(*======================================== 单电机控制标志位 Start ==================================*)								
	
	// 左臂单电机控制
	bAxis_LeftArm_Wrist_JogP			AT%MX0.0				:BOOL;			//左臂_腕电机_JOG正	
	bAxis_LeftArm_Wrist_JogN			AT%MX0.1				:BOOL;			//左臂_腕电机_JOG负
	bAxis_LeftArm_Left_JogP				AT%MX0.2				:BOOL;			//左臂_左电机_JOG正	
	bAxis_LeftArm_Left_JogN				AT%MX0.3				:BOOL;			//左臂_左电机_JOG负	
	bAxis_LeftArm_Right_JogP			AT%MX0.4				:BOOL;			//左臂_右电机_JOG正	
	bAxis_LeftArm_Right_JogN			AT%MX0.5				:BOOL;			//左臂_右电机_JOG负	
	bAxis_LeftArm_Lift_JogP				AT%MX0.6				:BOOL;			//左臂_升电机_JOG正	
	bAxis_LeftArm_Lift_JogN				AT%MX0.7				:BOOL;			//左臂_升电机_JOG负	

	// 右臂单电机控制
	bAxis_RightArm_Wrist_JogP			AT%MX1.6				:BOOL;			//右臂_腕电机_JOG正	
	bAxis_RightArm_Wrist_JogN			AT%MX1.7				:BOOL;			//右臂_腕电机_JOG负
	bAxis_RightArm_Left_JogP			AT%MX2.0				:BOOL;			//右臂_左电机_JOG正	
	bAxis_RightArm_Left_JogN			AT%MX2.1				:BOOL;			//右臂_左电机_JOG负	
	bAxis_RightArm_Right_JogP			AT%MX2.2				:BOOL;			//右臂_右电机_JOG正	
	bAxis_RightArm_Right_JogN			AT%MX2.3				:BOOL;			//右臂_右电机_JOG负	
	bAxis_RightArm_Lift_JogP			AT%MX2.4				:BOOL;			//右臂_升电机_JOG正	
	bAxis_RightArm_Lift_JogN			AT%MX2.5				:BOOL;			//右臂_升电机_JOG负			
	
	// 小龙门单电机控制
	bAxis_SmallGate_Left_JogP			AT%MX1.0				:BOOL;			//小门_左电机_JOG正
	bAxis_SmallGate_Left_JogN			AT%MX1.1				:BOOL;			//小门_左电机_JOG负
	bAxis_SmallGate_Right_JogP			AT%MX2.6				:BOOL;			//小门_右电机_JOG正
	bAxis_SmallGate_Right_JogN			AT%MX2.7				:BOOL;			//小门_右电机_JOG负	
	
	// 大龙门单电机控制
	bAxis_BigGate_Left_JogP				AT%MX1.2				:BOOL;			//大门_左电机_JOG正
	bAxis_BigGate_Left_JogN				AT%MX1.3				:BOOL;			//大门_左电机_JOG负
	bAxis_BigGate_Right_JogP			AT%MX3.0				:BOOL;			//大门_右电机_JOG正
	bAxis_BigGate_Right_JogN			AT%MX3.1				:BOOL;			//大门_右电机_JOG负	
	
	// 后龙门单电机控制
	bAxis_BackGate_Left_JogP			AT%MX1.4				:BOOL;			//后门_左电机_JOG正
	bAxis_BackGate_Left_JogN			AT%MX1.5				:BOOL;			//后门_左电机_JOG负
	bAxis_BackGate_Right_JogP			AT%MX3.2				:BOOL;			//后门_右电机_JOG正
	bAxis_BackGate_Right_JogN			AT%MX3.3				:BOOL;			//后门_右电机_JOG负	

(*===================================== 单电机控制标志位 End ========================================*)




	
(*===================================== 合成运动制标志位 Start ======================================*)		
	
	//左臂合成运动
	bLeftArm_Backward					AT%MX3.4				:BOOL;			//左臂_向后
	bLeftArm_Forward					AT%MX3.5				:BOOL;			//左臂_向前
	bLeftArm_Left						AT%MX3.6				:BOOL;			//左臂_向左
	bLeftArm_Right						AT%MX3.7				:BOOL;			//左臂_向右

	//右臂合成运动
	bRightArm_Backward					AT%MX4.0				:BOOL;			//左臂_向后
	bRightArm_Forward					AT%MX4.1				:BOOL;			//左臂_向前
	bRightArm_Left						AT%MX4.2				:BOOL;			//左臂_向左
	bRightArm_Right						AT%MX4.3				:BOOL;			//左臂_向右
	
	//小龙门合成运动jog
	bSmallGate_Up						AT%MX4.4				:BOOL;			//小门_升_jog
	bSmallGate_Down						AT%MX4.5				:BOOL;			//小门_降_jog
	
	//大龙门合成运动jog
	bBigGate_Up							AT%MX4.6				:BOOL;			//大门_升_jog
	bBigGate_Down						AT%MX4.7				:BOOL;			//大门_降_jog
	
	//后龙门合成运动jog
	bBackGate_Up						AT%MX5.0				:BOOL;			//后门_升_jog
	bBackGate_Down						AT%MX5.1				:BOOL;			//后门_降_jog
	
	//小龙门合成运动Abs
	bSmallGate_MoveAbs											:BOOL;			//小门_MoveAbs
	                                    	                                         
	//大龙门合成运动Abs                           	                                         
	bBigGate_MoveAbs											:BOOL;			//大门_MoveAbs
	                                    	                                         
	//后龙门合成运动Abs                           	                                         
	bBackGate_MoveAbs											:BOOL;			//后门_MoveAbs
	
(*===================================== 合成运动制标志位 End ========================================*)		






(*===================================== IO Input  ===================================================*)	
	bTeachBoxRemote						AT%IX0.0				:BOOL;			//示教盒旋钮Remote档
	bTeachBoxAuto						AT%IX0.1				:BOOL;			//示教盒旋钮Auto档
    bEmergencyStopBtn					AT%IX0.2				:BOOL;			//急停按钮
    bGreenBtn							AT%IX0.3				:BOOL;			//绿色按钮
    bYellowBtn							AT%IX0.4				:BOOL;			//黄色按钮
    bRedBtn								AT%IX0.5				:BOOL;			//红色按钮
    bRemoteCtrl_Online					AT%IX0.6				:BOOL;			//遥控器Online成功
	bRemoteCtrl_Up						AT%IX0.7				:BOOL;			//遥控器“上”按钮
	bRemoteCtrl_Down					AT%IX1.0				:BOOL;			//遥控器“下”按钮
	bRemoteCtrl_East					AT%IX1.1				:BOOL;			//遥控器“东”按钮
    bRemoteCtrl_West					AT%IX1.2				:BOOL;			//遥控器“西”按钮
    bRemoteCtrl_South					AT%IX1.3				:BOOL;			//遥控器“南”按钮
    bRemoteCtrl_North					AT%IX1.4				:BOOL;			//遥控器“北”按钮
    bRemoteCtrl_1btn					AT%IX1.5				:BOOL;			//遥控器“1”按钮
    bRemoteCtrl_2btn					AT%IX1.6				:BOOL;			//遥控器“2”按钮
	b_BackBeltCtrlBoxWarning			AT%IX1.7				:BOOL;			//长皮带变频器报警
	bLeftArm_Sucker1_Completed			AT%IX2.0				:BOOL;			//左吸盘组传感器1压力到达
	bLeftArm_Sucker2_Completed			AT%IX2.1				:BOOL;			//左吸盘组传感器2压力到达
    bLeftArm_Sucker3_Completed			AT%IX2.2				:BOOL;			//左吸盘组传感器3压力到达
    bLeftArm_Sucker4_Completed			AT%IX2.3				:BOOL;			//左吸盘组传感器4压力到达
    bLeftArm_Sucker5_Completed			AT%IX2.4				:BOOL;			//左吸盘组传感器5压力到达
    bLeftArm_Sucker6_Completed			AT%IX2.5				:BOOL;			//左吸盘组传感器6压力到达
    bLeftArm_Sucker7_Completed			AT%IX2.6				:BOOL;			//左吸盘组传感器7压力到达
	bLeftArm_Sucker8_Completed			AT%IX2.7				:BOOL;			//左吸盘组传感器8压力到达
	bRightArm_Sucker1_Completed			AT%IX3.0				:BOOL;			//右吸盘组传感器1压力到达
	bRightArm_Sucker2_Completed			AT%IX3.1				:BOOL;			//右吸盘组传感器2压力到达
	bRightArm_Sucker3_Completed			AT%IX3.2				:BOOL;			//右吸盘组传感器3压力到达
	bRightArm_Sucker4_Completed			AT%IX3.3				:BOOL;			//右吸盘组传感器4压力到达
	bRightArm_Sucker5_Completed			AT%IX3.4				:BOOL;			//右吸盘组传感器5压力到达
	bRightArm_Sucker6_Completed			AT%IX3.5				:BOOL;			//右吸盘组传感器6压力到达
	bRightArm_Sucker7_Completed			AT%IX3.6				:BOOL;			//右吸盘组传感器7压力到达
	bRightArm_Sucker8_Completed			AT%IX3.7				:BOOL;			//右吸盘组传感器8压力到达
	bCrash_Sensor_Front					AT%IX4.0				:BOOL;			//前防撞条动作
	bCrash_Sensor_Back					AT%IX4.1				:BOOL;			//后防撞条动作	
	bPumpPhaseSequenceProtectionOK		AT%IX5.0				:bool;			//气泵相序保护器OK标志位
(*===================================== IO Input ====================================================*)	





(*===================================== 电磁阀控制标志位 Start ======================================*)	
	
	//左臂电磁阀
	bLeftArm_SV1						AT%QX2.0				:BOOL;			//左臂_电磁阀1
	bLeftArm_SV2						AT%QX2.1				:BOOL;			//左臂_电磁阀2	
	bLeftArm_SV3						AT%QX2.2				:BOOL;			//左臂_电磁阀3
	bLeftArm_SV4						AT%QX2.3				:BOOL;			//左臂_电磁阀4
	bLeftArm_SV5						AT%QX2.4				:BOOL;			//左臂_电磁阀5
	bLeftArm_SV6						AT%QX2.5				:BOOL;			//左臂_电磁阀6
	bLeftArm_SV7						AT%QX2.6				:BOOL;			//左臂_电磁阀7	
	bLeftArm_SV8						AT%QX2.7				:BOOL;			//左臂_电磁阀8
	
	//左臂电磁阀
	bRightArm_SV1						AT%QX3.0				:BOOL;			//右臂_电磁阀1
	bRightArm_SV2						AT%QX3.1				:BOOL;			//右臂_电磁阀2	
	bRightArm_SV3						AT%QX3.2				:BOOL;			//右臂_电磁阀3
	bRightArm_SV4						AT%QX3.3				:BOOL;			//右臂_电磁阀4
	bRightArm_SV5						AT%QX3.4				:BOOL;			//右臂_电磁阀5
	bRightArm_SV6						AT%QX3.5				:BOOL;			//右臂_电磁阀6
	bRightArm_SV7						AT%QX3.6				:BOOL;			//右臂_电磁阀7	
	bRightArm_SV8						AT%QX3.7				:BOOL;			//右臂_电磁阀8
	
	aLeftArm_SV_Array					:ARRAY[1..8] OF BOOL:=[bLeftArm_SV1,
                                                               bLeftArm_SV2,
                                                               bLeftArm_SV3,
                                                               bLeftArm_SV4,
                                                               bLeftArm_SV5,
                                                               bLeftArm_SV6,
                                                               bLeftArm_SV7,
                                                               bLeftArm_SV8	
																];
																
	aRightArm_SV_Array					:ARRAY[1..8] OF BOOL:=[bRightArm_SV1,
                                                               bRightArm_SV2,
                                                               bRightArm_SV3,
                                                               bRightArm_SV4,
                                                               bRightArm_SV5,
                                                               bRightArm_SV6,
                                                               bRightArm_SV7,
                                                               bRightArm_SV8	
																];

	//左臂电磁阀_示教盒标志位
	bLeftArm_SV1_TBox						AT%MX7.0				:BOOL;			//左臂_电磁阀1_示教盒标志位
	bLeftArm_SV2_TBox						AT%MX7.1				:BOOL;			//左臂_电磁阀2_示教盒标志位	
	bLeftArm_SV3_TBox						AT%MX7.2				:BOOL;			//左臂_电磁阀3_示教盒标志位
	bLeftArm_SV4_TBox						AT%MX7.3				:BOOL;			//左臂_电磁阀4_示教盒标志位
	bLeftArm_SV5_TBox						AT%MX7.4				:BOOL;			//左臂_电磁阀5_示教盒标志位
	bLeftArm_SV6_TBox						AT%MX7.5				:BOOL;			//左臂_电磁阀6_示教盒标志位
	bLeftArm_SV7_TBox						AT%MX7.6				:BOOL;			//左臂_电磁阀7_示教盒标志位	
	bLeftArm_SV8_TBox						AT%MX7.7				:BOOL;			//左臂_电磁阀8_示教盒标志位
	
	//右臂电磁阀_示教盒标志位
	bRightArm_SV1_TBox						AT%MX8.0				:BOOL;			//右臂_电磁阀1_示教盒标志位
	bRightArm_SV2_TBox						AT%MX8.1				:BOOL;			//右臂_电磁阀2_示教盒标志位
	bRightArm_SV3_TBox						AT%MX8.2				:BOOL;			//右臂_电磁阀3_示教盒标志位
	bRightArm_SV4_TBox						AT%MX8.3				:BOOL;			//右臂_电磁阀4_示教盒标志位
	bRightArm_SV5_TBox						AT%MX8.4				:BOOL;			//右臂_电磁阀5_示教盒标志位
	bRightArm_SV6_TBox						AT%MX8.5				:BOOL;			//右臂_电磁阀6_示教盒标志位
	bRightArm_SV7_TBox						AT%MX8.6				:BOOL;			//右臂_电磁阀7_示教盒标志位
	bRightArm_SV8_TBox						AT%MX8.7				:BOOL;			//右臂_电磁阀8_示教盒标志位

	
	//左臂电磁阀_示教盒上位机
	bLeftArm_SV1_UpperUI											:BOOL;			//左臂_电磁阀1_上位机标志位
	bLeftArm_SV2_UpperUI											:BOOL;			//左臂_电磁阀2_上位机标志位	
	bLeftArm_SV3_UpperUI											:BOOL;			//左臂_电磁阀3_上位机标志位
	bLeftArm_SV4_UpperUI											:BOOL;			//左臂_电磁阀4_上位机标志位
	bLeftArm_SV5_UpperUI											:BOOL;			//左臂_电磁阀5_上位机标志位
	bLeftArm_SV6_UpperUI											:BOOL;			//左臂_电磁阀6_上位机标志位
	bLeftArm_SV7_UpperUI											:BOOL;			//左臂_电磁阀7_上位机标志位	
	bLeftArm_SV8_UpperUI											:BOOL;			//左臂_电磁阀8_上位机标志位
	                                            	                                            
	//左臂电磁阀_示教盒上位机                              	                                            
	bRightArm_SV1_UpperUI											:BOOL;			//右臂_电磁阀1_上位机标志位
	bRightArm_SV2_UpperUI											:BOOL;			//右臂_电磁阀2_上位机标志位
	bRightArm_SV3_UpperUI											:BOOL;			//右臂_电磁阀3_上位机标志位
	bRightArm_SV4_UpperUI											:BOOL;			//右臂_电磁阀4_上位机标志位
	bRightArm_SV5_UpperUI											:BOOL;			//右臂_电磁阀5_上位机标志位
	bRightArm_SV6_UpperUI											:BOOL;			//右臂_电磁阀6_上位机标志位
	bRightArm_SV7_UpperUI											:BOOL;			//右臂_电磁阀7_上位机标志位
	bRightArm_SV8_UpperUI											:BOOL;			//右臂_电磁阀8_上位机标志位


	
(*===================================== 电磁阀控制标志位 End ========================================*)	







(*===================================== 灯光 Start ========================================*)
	
	bTriColorLed_Green_Enable					AT%QX0.0				:BOOL;			//三色灯-绿色-点亮
	bTriColorLed_Yellow_Enable					AT%QX0.1				:BOOL;			//三色灯-黄色-点亮
	bTriColorLed_Red_Enable						AT%QX0.2				:BOOL;			//三色灯-红色-点亮
	bBtnLed_Green_Enable						AT%QX0.3				:BOOL;			//按钮灯-绿色-点亮
	bBtnLed_Yellow_Enable						AT%QX0.4				:BOOL;			//按钮灯-黄色-点亮
	bBtnLed_Red_Enable							AT%QX0.5				:BOOL;			//按钮灯-红色-点亮
	bFrontLight_Left_Enable						AT%QX0.6				:BOOL;			//前部照明灯-左-点亮
	bFrontLight_Right_Enable					AT%QX0.7				:BOOL;			//前部照明灯-右-点亮	
	
(*===================================== 灯光 End ==========================================*)	





(*===================================== 真空泵 Start ========================================*)
	
	bPumpMotor_Enable					AT%QX1.0				:BOOL;			//真空泵电机上电
	bPumpMotor_Enable_TBox				AT%MX9.4				:BOOL;			//真空泵电机上电_示教盒标志位
	bPumpMotor_Enable_UpperUI									:BOOL;			//真空泵电机上电_上位机标志位
	
(*===================================== 真空泵 End ==========================================*)





(*===================================== 滚筒控制标志位 Start ========================================*)
	
	bAxis_GunTong_Back					AT%QX1.1				:BOOL;			//后滚筒_电机
	bAxis_GunTong_Left					AT%QX1.2				:BOOL;			//左滚筒_电机
	bAxis_GunTong_Right					AT%QX1.3				:BOOL;			//右滚筒_电机
	bAxis_GunTong_Middle				AT%QX1.4				:BOOL;			//中滚筒_电机

(*===================================== 滚筒控制标志位 End ==========================================*)





(*===================================== 示教盒相关 Start ============================================*)	
	
//	bTeachBox_Stop						AT%MX5.2				:BOOL;			//示教盒STOP键
//	bTeachBox_Run						AT%MX5.3				:BOOL;			//示教盒Run键
//	bTeachBox_Hand00					AT%MX5.4				:BOOL;			//示教盒HAND00键
//	bTeachBox_Hand01					AT%MX5.5				:BOOL;			//示教盒HAND01键
//	bTeachBox_Led1						AT%MX6.0				:BOOL;			//示教盒LED1点亮
//	bTeachBox_Led2						AT%MX6.1				:BOOL;			//示教盒LED2点亮
//	bTeachBox_Buzzer_continuous			AT%MX6.2				:BOOL;			//示教盒蜂鸣器长蜂鸣	
//	bTeachBox_Buzzer_Short				AT%MX6.2				:BOOL;			//示教盒蜂鸣器短蜂鸣

(*===================================== 示教盒相关 End ==============================================*)	






(*===================================== 运行速度设置区 Start ========================================*)	
	
//	//手动模式速度及加速度设置
//	fManualCtrl_Velo					AT%MD20					:REAL;			//手动控制_运行速度
//	fManualCtrl_Acc						AT%MD24					:REAL;			//手动控制_运行速度
	
//	//自动模式速度及加速度设置
//	fAutoCtrl_Velo						AT%MD28					:REAL;			//自动控制_运行速度
//	fAutoCtrl_Acc						AT%MD32					:REAL;			//自动控制_运行速度			

(*===================================== 运行速度设置区 End ==========================================*)	




(*====================================== 状态显示字段 Start =========================================*)	
	
//	//左臂电机状态
//	fAxis_LeftArm_Wrist_ActPos			AT%MD100				:REAL;			//左臂_腕电机_实时位置
//	fAxis_LeftArm_Wrist_ActVelo			AT%MD104				:REAL;			//左臂_腕电机_实时速度
//	fAxis_LeftArm_Wrist_ActTorq			AT%MD108				:REAL;			//左臂_腕电机_实时力矩	
//	fAxis_LeftArm_Left_ActPos			AT%MD112				:REAL;			//左臂_左电机_实时位置
//	fAxis_LeftArm_Left_ActVelo			AT%MD116				:REAL;			//左臂_左电机_实时速度
//	fAxis_LeftArm_Left_ActTorq			AT%MD120				:REAL;			//左臂_左电机_实时力矩		
//	fAxis_LeftArm_Right_ActPos			AT%MD124				:REAL;			//左臂_右电机_实时位置
//	fAxis_LeftArm_Right_ActVelo			AT%MD128				:REAL;			//左臂_右电机_实时速度
//	fAxis_LeftArm_Right_ActTorq			AT%MD132				:REAL;			//左臂_右电机_实时力矩
//	fAxis_LeftArm_Lift_ActPos			AT%MD136				:REAL;			//左臂_升电机_实时位置
//	fAxis_LeftArm_Lift_ActVelo			AT%MD140				:REAL;			//左臂_升电机_实时速度
//	fAxis_LeftArm_Lift_ActTorq			AT%MD144				:REAL;			//左臂_升电机_实时力矩

//	//右臂电机状态
//	fAxis_RightArm_Wrist_ActPos			AT%MD184				:REAL;			//右臂_腕电机_实时位置
//	fAxis_RightArm_Wrist_ActVelo		AT%MD188				:REAL;			//右臂_腕电机_实时速度
//	fAxis_RightArm_Wrist_ActTorq		AT%MD192				:REAL;			//右臂_腕电机_实时力矩	
//	fAxis_RightArm_Left_ActPos			AT%MD196				:REAL;			//右臂_左电机_实时位置
//	fAxis_RightArm_Left_ActVelo			AT%MD200				:REAL;			//右臂_左电机_实时速度
//	fAxis_RightArm_Left_ActTorq			AT%MD204				:REAL;			//右臂_左电机_实时力矩		
//	fAxis_RightArm_Right_ActPos			AT%MD208				:REAL;			//右臂_右电机_实时位置
//	fAxis_RightArm_Right_ActVelo		AT%MD212				:REAL;			//右臂_右电机_实时速度
//	fAxis_RightArm_Right_ActTorq		AT%MD216				:REAL;			//右臂_右电机_实时力矩
//	fAxis_RightArm_Lift_ActPos			AT%MD220				:REAL;			//右臂_升电机_实时位置
//	fAxis_RightArm_Lift_ActVelo			AT%MD224				:REAL;			//右臂_升电机_实时速度
//	fAxis_RightArm_Lift_ActTorq			AT%MD228				:REAL;			//右臂_升电机_实时力矩				
	
//	//小龙门电机状态
//	fAxis_SmallGate_Left_ActPos			AT%MD148				:REAL;			//小龙门_左电机_实时位置
//	fAxis_SmallGate_Left_ActVelo		AT%MD152				:REAL;			//小龙门_左电机_实时速度
//	fAxis_SmallGate_Left_ActTorq		AT%MD156				:REAL;			//小龙门_左电机_实时力矩
//	fAxis_SmallGate_Right_ActPos		AT%MD232				:REAL;			//小龙门_右电机_实时位置
//	fAxis_SmallGate_Right_ActVelo		AT%MD236				:REAL;			//小龙门_右电机_实时速度
//	fAxis_SmallGate_Right_ActTorq		AT%MD240				:REAL;			//小龙门_右电机_实时力矩

//	//大龙门电机状态
//	fAxis_BigGate_Left_ActPos			AT%MD160				:REAL;			//大龙门_左电机_实时位置
//	fAxis_BigGate_Left_ActVelo			AT%MD164				:REAL;			//大龙门_左电机_实时速度
//	fAxis_BigGate_Left_ActTorq			AT%MD168				:REAL;			//大龙门_左电机_实时力矩
//	fAxis_BigGate_Right_ActPos			AT%MD244				:REAL;			//大龙门_右电机_实时位置
//	fAxis_BigGate_Right_ActVelo			AT%MD248				:REAL;			//大龙门_右电机_实时速度
//	fAxis_BigGate_Right_ActTorq			AT%MD252				:REAL;			//大龙门_右电机_实时力矩

//	//后龙门电机状态
//	fAxis_BackGate_Left_ActPos			AT%MD172				:REAL;			//后龙门_左电机_实时位置
//	fAxis_BackGate_Left_ActVelo			AT%MD176				:REAL;			//后龙门_左电机_实时速度
//	fAxis_BackGate_Left_ActTorq			AT%MD180				:REAL;			//后龙门_左电机_实时力矩
//	fAxis_BackGate_Right_ActPos			AT%MD256				:REAL;			//后龙门_右电机_实时位置
//	fAxis_BackGate_Right_ActVelo		AT%MD260				:REAL;			//后龙门_右电机_实时速度
//	fAxis_BackGate_Right_ActTorq		AT%MD264				:REAL;			//后龙门_右电机_实时力矩
	
	
	

(*====================================== 状态显示字段  End ==========================================*)	





END_VAR

// ---- GVLs/Robot_Motor.TcGVL
//{attribute 'qualified_only'}
VAR_GLOBAL
	
(*======================================== 机器人各轴定义 Start ==========================================*)
	// 左臂电机
	axis_LeftArm_Wrist											:AXIS_REF;			//左臂_腕电机	
	axis_LeftArm_Left											:AXIS_REF;			//左臂_左电机
	axis_LeftArm_Right											:AXIS_REF;			//左臂_右电机	
	axis_LeftArm_Lift											:AXIS_REF;			//左臂_升电机	

	// 右臂电机
	axis_RightArm_Wrist											:AXIS_REF;			//右臂_腕电机	
	axis_RightArm_Left											:AXIS_REF;			//右臂_左电机
	axis_RightArm_Right											:AXIS_REF;			//右臂_右电机
	axis_RightArm_Lift											:AXIS_REF;			//右臂_升电机
	
	// 小龙门电机
	axis_SmallGate_Left											:AXIS_REF;			//小门_左电机
	axis_SmallGate_Right										:AXIS_REF;			//小门_右电机

	
	// 大龙门单电机
	axis_BigGate_Left											:AXIS_REF;			//大门_左电机
	axis_BigGate_Right											:AXIS_REF;			//大门_右电机
	
	// 后龙门单电机
	axis_BackGate_Left											:AXIS_REF;			//后门_左电机
	axis_BackGate_Right											:AXIS_REF;			//后门_右电机
	
	// 右轮
	axis_RightWheel_Steer										:AXIS_REF;			
	axis_RightWheel_Walk										:AXIS_REF;	
	
	// 左轮
	axis_LeftWheel_Steer										:AXIS_REF;			
	axis_LeftWheel_Walk											:AXIS_REF;		
	

	nAxisNum							: USINT:=18;						// 轴组管理的轴的数量
	
	// 轴组
	aAxisGroup							: ARRAY[1..24] OF POINTER TO AXIS_REF :=[
																	  ADR(axis_LeftArm_Wrist),
																	  ADR(axis_LeftArm_Left),
																	  ADR(axis_LeftArm_Right),
																	  ADR(axis_LeftArm_Lift),
																	  ADR(axis_RightArm_Wrist),
																	  ADR(axis_RightArm_Left),
																	  ADR(axis_RightArm_Right),
																	  ADR(axis_RightArm_Lift),
																	  ADR(axis_SmallGate_Left),
																	  ADR(axis_SmallGate_Right),
																	  ADR(axis_BigGate_Left),
																	  ADR(axis_BigGate_Right),
																	  ADR(axis_BackGate_Left),
																	  ADR(axis_BackGate_Right),
																	  ADR(axis_RightWheel_Steer),
																	  ADR(axis_RightWheel_Walk),
																	  ADR(axis_LeftWheel_Steer),
																	  ADR(axis_LeftWheel_Walk)
																	 ];			


	

(*======================================== 机器人各轴定义 End =============================================*)	




(*======================================== 机器人各轴力矩 Start =============================================*)	
	
	axis_RightArm_Left_Torque				AT%I*				:INT;
	axis_RightArm_Right_Torque				AT%I*				:INT;
	axis_RightArm_Wrist_Torque				AT%I*				:INT;
	axis_RightArm_Lift_Torque				AT%I*				:INT;
	axis_LeftArm_Left_Torque				AT%I*				:INT;
	axis_LeftArm_Right_Torque				AT%I*				:INT;
	axis_LeftArm_Wrist_Torque				AT%I*				:INT;
	axis_LeftArm_Lift_Torque				AT%I*				:INT;	
	axis_SmallGate_Left_Torque				AT%I*				:INT;
	axis_SmallGate_Right_Torque				AT%I*				:INT;
	axis_BigGate_Left_Torque				AT%I*				:INT;
	axis_BigGate_Right_Torque				AT%I*				:INT;	
	axis_BackGate_Left_Torque				AT%I*				:INT;
	axis_BackGate_Right_Torque				AT%I*				:INT;	
	
(*======================================== 机器人各轴力矩  End =============================================*)	


	

(*======================================== 机器人各轴 MC_Power定义 Start ==================================*)
	
	// 左臂电机
	axis_LeftArm_Wrist_Power									:MC_Power;			//左臂_腕电机Power功能块	
	axis_LeftArm_Left_Power										:MC_Power;			//左臂_左电机Power功能块
	axis_LeftArm_Right_Power									:MC_Power;			//左臂_右电机Power功能块
	axis_LeftArm_Lift_Power										:MC_Power;			//左臂_升电机Power功能块

	// 右臂电机
	axis_RightArm_Wrist_Power									:MC_Power;			//右臂_腕电机Power功能块	
	axis_RightArm_Left_Power									:MC_Power;			//右臂_左电机Power功能块
	axis_RightArm_Right_Power									:MC_Power;			//右臂_右电机Power功能块
	axis_RightArm_Lift_Power									:MC_Power;			//右臂_升电机Power功能块
	
	// 小龙门电机
	axis_SmallGate_Left_Power									:MC_Power;			//小门_左电机Power功能块
	axis_SmallGate_Right_Power									:MC_Power;			//小门_右电机Power功能块

	// 大龙门单电机
	axis_BigGate_Left_Power										:MC_Power;			//大门_左电机Power功能块
	axis_BigGate_Right_Power									:MC_Power;			//大门_右电机Power功能块
	
	// 后龙门单电机
	axis_BackGate_Left_Power									:MC_Power;			//后门_左电机Power功能块
	axis_BackGate_Right_Power									:MC_Power;			//后门_右电机Power功能块
	
	// 右轮
	axis_RightWheel_Steer_Power									:MC_Power;
	axis_RightWheel_Walk_Power									:MC_Power;
	
	// 左轮
	axis_LeftWheel_Steer_Power									:MC_Power;
	axis_LeftWheel_Walk_Power									:MC_Power;	

	// 左臂电机
	axis_LeftArm_Wrist_Power_Output									:ST_McOutputs;			//左臂_腕电机状态	
	axis_LeftArm_Left_Power_Output									:ST_McOutputs;			//左臂_左电机状态
	axis_LeftArm_Right_Power_Output									:ST_McOutputs;			//左臂_右电机状态
	axis_LeftArm_Lift_Power_Output									:ST_McOutputs;			//左臂_升电机状态

	// 右臂电机
	axis_RightArm_Wrist_Power_Output								:ST_McOutputs;			//右臂_腕电机Power功能块	
	axis_RightArm_Left_Power_Output									:ST_McOutputs;			//右臂_左电机Power功能块
	axis_RightArm_Right_Power_Output								:ST_McOutputs;			//右臂_右电机Power功能块
	axis_RightArm_Lift_Power_Output									:ST_McOutputs;			//右臂_升电机Power功能块
	
	// 小龙门电机
	axis_SmallGate_Left_Power_Output								:ST_McOutputs;			//小门_左电机Power功能块
	axis_SmallGate_Right_Power_Output								:ST_McOutputs;			//小门_右电机Power功能块

	// 大龙门单电机
	axis_BigGate_Left_Power_Output									:ST_McOutputs;			//大门_左电机Power功能块
	axis_BigGate_Right_Power_Output									:ST_McOutputs;			//大门_右电机Power功能块
	
	// 后龙门单电机
	axis_BackGate_Left_Power_Output									:ST_McOutputs;			//后门_左电机Power功能块
	axis_BackGate_Right_Power_Output								:ST_McOutputs;			//后门_右电机Power功能块	
	
	// 右轮
	axis_RightWheel_Steer_Power_Output									:ST_McOutputs;
	axis_RightWheel_Walk_Power_Output									:ST_McOutputs;
	
	// 左轮
	axis_LeftWheel_Steer_Power_Output									:ST_McOutputs;
	axis_LeftWheel_Walk_Power_Output									:ST_McOutputs;
	
(*======================================== 机器人各轴 MC_Power定义 Start ==================================*)





(*======================================== 机器人各轴 MC_Reset定义 Start ==================================*)

	// 左臂电机
	axis_LeftArm_Wrist_Reset									:MC_Reset;			//左臂_腕电机Power功能块	
	axis_LeftArm_Left_Reset										:MC_Reset;			//左臂_左电机Power功能块
	axis_LeftArm_Right_Reset									:MC_Reset;			//左臂_右电机Power功能块
	axis_LeftArm_Lift_Reset										:MC_Reset;			//左臂_升电机Power功能块

	// 右臂电机
	axis_RightArm_Wrist_Reset									:MC_Reset;			//右臂_腕电机Power功能块	
	axis_RightArm_Left_Reset									:MC_Reset;			//右臂_左电机Power功能块
	axis_RightArm_Right_Reset									:MC_Reset;			//右臂_右电机Power功能块
	axis_RightArm_Lift_Reset									:MC_Reset;			//右臂_升电机Power功能块
	
	// 小龙门电机
	axis_SmallGate_Left_Reset									:MC_Reset;			//小门_左电机Power功能块
	axis_SmallGate_Right_Reset									:MC_Reset;			//小门_右电机Power功能块

	// 大龙门单电机
	axis_BigGate_Left_Reset										:MC_Reset;			//大门_左电机Power功能块
	axis_BigGate_Right_Reset									:MC_Reset;			//大门_右电机Power功能块
	
	// 后龙门单电机
	axis_BackGate_Left_Reset									:MC_Reset;			//后门_左电机Power功能块
	axis_BackGate_Right_Reset									:MC_Reset;			//后门_右电机Power功能块

	// 右轮
	axis_RightWheel_Steer_Reset									:MC_Reset;
	axis_RightWheel_Walk_Reset									:MC_Reset;
	
	// 左轮
	axis_LeftWheel_Steer_Reset									:MC_Reset;
	axis_LeftWheel_Walk_Reset									:MC_Reset;	

(*======================================== 机器人各轴 MC_Reset定义 End ==================================*)


	

(*======================================== 机器人各轴 MC_Jog定义 Start ==================================*)
	
	bJogFast												:BOOL;									// 快速Jog标志位
	aAxis_Jog_Speed											:ARRAY[0..1] OF LREAL:=[1,5];			// JOG speed

	// 左臂电机
	axis_LeftArm_Wrist_Jog									:MC_Jog;			//左臂_腕电机Jog功能块	
	axis_LeftArm_Left_Jog									:MC_Jog;			//左臂_左电机Jog功能块
	axis_LeftArm_Right_Jog									:MC_Jog;			//左臂_右电机Jog功能块
	axis_LeftArm_Lift_Jog									:MC_Jog;			//左臂_升电机Jog功能块
	
	// 右臂电机
	axis_RightArm_Wrist_Jog									:MC_Jog;			//右臂_腕电机Jog功能块	
	axis_RightArm_Left_Jog									:MC_Jog;			//右臂_左电机Jog功能块
	axis_RightArm_Right_Jog									:MC_Jog;			//右臂_右电机Jog功能块
	axis_RightArm_Lift_Jog									:MC_Jog;			//右臂_升电机Jog功能块
	
	// 小龙门电机
	axis_SmallGate_Left_Jog									:MC_Jog;			//小门_左电机Jog功能块
	axis_SmallGate_Right_Jog								:MC_Jog;			//小门_右电机Jog功能块
	
	// 大龙门单电机
	axis_BigGate_Left_Jog									:MC_Jog;			//大门_左电机Jog功能块
	axis_BigGate_Right_Jog									:MC_Jog;			//大门_右电机Jog功能块
	
	// 后龙门单电机
	axis_BackGate_Left_Jog									:MC_Jog;			//后门_左电机Jog功能块
	axis_BackGate_Right_Jog									:MC_Jog;			//后门_右电机Jog功能块

	// 右轮
	axis_RightWheel_Steer_Jog								:MC_Jog;
	axis_RightWheel_Walk_Jog								:MC_Jog;
	
	// 左轮
	axis_LeftWheel_Steer_Jog								:MC_Jog;
	axis_LeftWheel_Walk_Jog									:MC_Jog;
	
	

(*======================================== 机器人各轴 MC_Jog定义 End =====================================*)




(*======================================== 机器人各轴 MC_MoveAbs定义 Start ==================================*)
	
